	WheelB.ControlFeedbackSign := 1.0;
	WheelB.CarouselSign := -1.0;
	WheelB.StandardSign := 1.0;
	WheelB.DriveWheel := FALSE;
	WheelB.InnerFlag := TRUE;
	WheelB.WheelDirection := -1.0;
	WheelB.IndependentWheels := TRUE;

	WheelC.ControlFeedbackSign := 1.0;
	WheelC.CarouselSign := 1.0;
	WheelC.StandardSign := -1.0;
	WheelC.DriveWheel := TRUE;
	WheelC.InnerFlag := TRUE;
	WheelC.WheelDirection := -1.0;
	WheelC.IndependentWheels := TRUE;

	WheelD.ControlFeedbackSign := 1.0;
	WheelD.CarouselSign := -1.0;
	WheelD.StandardSign := -1.0;
	WheelD.DriveWheel := TRUE;
	WheelD.InnerFlag := FALSE;
	WheelD.WheelDirection := 1.0;
	WheelD.IndependentWheels := TRUE;
{END_IF}

lFunctionalMode := cFunctionalModeAny;

lMode REF= lSteerMode4WS;

lTargetAngleUpdateTimer.Period := cTargetAngleUpdatePeriod;
lTargetAngleUpdateTimer.Enable := TRUE;
lTargetAngleUpdateTimer.initialize();

                
END_METHOD

METHOD operator
                  requestSteerMode(gSystemPrimary.UInterface.SteerModeRequest);

lInput.InputAsPercentage := gSystemPrimary.UInterface.Steer;
lInput.operator();

SUPER^.operator();

lZeroTargetAngleSwitch.Value := gSystemPrimary.UInterface.ZeroSteerTargetAngle;
lZeroTargetAngleSwitch.operator();

IF (lEnableRelativeSteering) THEN
	lRegisterActive := TRUE;

	IF ((lZeroTargetAngleSwitch.Value) AND (lEnableZeroTargetAngleSwitch)) THEN
		zeroTargetAngle();
	END_IF

	lTargetAngleShift := lInput.Value;
ELSE
	lRegisterActive := TRUE;
	
	IF (lZeroTargetAngleSwitch.Value) THEN
		gSystemPrimary.Active.registerActive();
	END_IF
	
	IF (gSystemPrimary.Active.Allow) THEN
		lRequestedAbsoluteTargetAngle := lInput.Value;
		
		IF (lRequestedAbsoluteTargetAngle>=Mode.SteerAngleMaximum) THEN
			lRequestedAbsoluteTargetAngle := Mode.SteerAngleMaximum;
		END_IF
		IF (lRequestedAbsoluteTargetAngle<=Mode.SteerAngleMinimum) THEN
			lRequestedAbsoluteTargetAngle := Mode.SteerAngleMinimum;
		END_IF
	
		lTargetAngleShift := (lRequestedAbsoluteTargetAngle - lTargetAngle.Value) * cSteerAbsoluteShiftFactor;
	ELSE
		lTargetAngleShift := 0.0;	
	END_IF
	
	IF (lTargetAngleShift<-1.0) THEN
		lTargetAngleShift := -1.0;
	END_IF
	IF (lTargetAngleShift>1.0) THEN
		lTargetAngleShift := 1.0;
	END_IF
END_IF

updateTargetAngle();
checkWheelStates();

lWheelA.operator();
lWheelB.operator();
lWheelC.operator();
lWheelD.operator();

IF (lStalledSubSystems) THEN
	IF (NOT(lStalledSubSystemsPrevious)) THEN
		lStallClearPreCondition := NOT(InputPresentAny);
		lStallClearPreConditionCleared := FALSE;
	END_IF
	
	lStalled := TRUE;
END_IF

IF (lStalled) THEN
	lStallClearPreConditionCleared := (((InputPresentAny) AND (lStallClearPreCondition)) OR
		((NOT(InputPresentAny)) AND (NOT(lStallClearPreCondition))));
		
	lStalled := (NOT((gSystemPrimary.Travel.InputPresentAny) OR
		((InputPresentAny) AND
		(lStallClearPreConditionCleared))));
END_IF

IF (NOT(lStalled)) THEN
	WheelA.Throttle.clearStalled();
	WheelB.Throttle.clearStalled();
	WheelC.Throttle.clearStalled();
	WheelD.Throttle.clearStalled();
END_IF

                
END_METHOD

METHOD requestSteerMode : t_steer_mode_diagnostic
  VAR_INPUT
    requestedSteerMode : t_steer_mode;
  END_VAR
  VAR
    angle : REAL;
  END_VAR
                  IF (requestedSteerMode=cSteerModeNone) THEN
	RETURN;
END_IF

lSteerModeDiagnostic := cSteerModeDiagnosticOK;

IF (Mode.matches(requestedSteerMode)) THEN
	// essentially re-initializes to this steering mode
	angle := Mode.getInitialTargetAngle(lTargetAngle.Value,requestedSteerMode);
	IF (lTargetAngle.Value<>angle) THEN
		lTargetAngle.Value := angle;
		
		lWheelA.ModeChange := TRUE;
		lWheelB.ModeChange := TRUE;
		lWheelC.ModeChange := TRUE;
		lWheelD.ModeChange := TRUE;
		
		IF (lEnableSequentialModeChange) THEN
			lWheelA.ModeChangeDisableControl := FALSE;
			lWheelB.ModeChangeDisableControl := TRUE;
			lWheelC.ModeChangeDisableControl := TRUE;
			lWheelD.ModeChangeDisableControl := TRUE;
		END_IF
	END_IF
	
	requestSteerMode := lSteerModeDiagnostic;
	RETURN;
END_IF

IF (NOT(checkModeEnabled(requestedSteerMode))) THEN
	lSteerModeDiagnostic := cSteerModeDiagnosticNotEnabled;
	//gMessageManager.register(lCode:=cMCAdviseSteerModeIllegalRequest);

	requestSteerMode := lSteerModeDiagnostic;
	RETURN;
END_IF
	
IF ((lEnableOperatingModeLockOnSteerModeChange) AND
	(gSystemPrimary.OperatingMode.lock(cOperatingModeLockPeriod)<>cOperatingModeLocked)) THEN
	lSteerModeDiagnostic := cSteerModeDiagnosticUnableToLockDrive;
	//gMessageManager.register(lCode:=cMCAdviseSteerModeUnableToLockDrive);
	
	requestSteerMode := lSteerModeDiagnostic;
	RETURN;
END_IF

lMode.leave();
lMode REF= getMode(requestedSteerMode);
lSteerModeDiagnostic := cSteerModeDiagnosticChanging;

lTargetAngle.Value := Mode.getInitialTargetAngle(0.0,requestedSteerMode);

lWheelA.ModeChange := TRUE;
lWheelB.ModeChange := TRUE;
lWheelC.ModeChange := TRUE;
lWheelD.ModeChange := TRUE;

IF (lEnableSequentialModeChange) THEN // foobar apollo issue remaining - not all wheels are moving at the same time during mode changes, but could be spurious due to stalling
	lWheelA.ModeChangeDisableControl := FALSE;
	lWheelB.ModeChangeDisableControl := TRUE;
	lWheelC.ModeChangeDisableControl := TRUE;
	lWheelD.ModeChangeDisableControl := TRUE;
END_IF

// checkWheelStates();

                
END_METHOD

METHOD setCarouselAngle
                  lCarouselAngle := ATAN(lSteerWheelBase/lSteerWheelTrack);

                
END_METHOD

METHOD toggleSteerMode
                  CASE lMode.Mode OF
	cSteerModeNone:
		requestSteerMode(cSteerMode4WS);
	cSteerMode4WS:
		requestSteerMode(cSteerModeLateral);
	cSteerModeLateral:
		requestSteerMode(cSteerModeCarousel);
	cSteerModeCarousel:
		requestSteerMode(cSteerMode4WS);
END_CASE

                
END_METHOD

METHOD updateTargetAngle
                  IF (lEnableUpdateTimer) THEN
	lTargetAngleUpdateTimer.operator();
	IF (NOT(lTargetAngleUpdateTimer.lExpired)) THEN
		RETURN;
	END_IF
	lTargetAngleUpdateTimer.reset();
END_IF

IF (lTargetAngleShift=0.0) THEN
	IF (lEnableDerivedTargetAngleIncrement) THEN
		lTargetAngleIncrementDerivedPost := lTargetAngleIncrementDerived;
		
		IF (((lTargetAngleIncrementDerived>0) AND
			(ABS(lCurrentPositiveDelta)>cSteerAngleMaxDerivedUpdateDelta)) OR
			((lTargetAngleIncrementDerived<0) AND
			(ABS(lCurrentNegativeDelta)>cSteerAngleMaxDerivedUpdateDelta))) THEN
			lTargetAngleIncrementDerivedPost := 0.0;
		END_IF
			
		lTargetAngle.Value := lTargetAngle.Value + lTargetAngleIncrementDerivedPost;

		//lTargetAngleIncrementDerived := 0.0;
	END_IF
ELSE
	lTargetAngleIncrement := 0;

	IF (lTargetAngleShift>0) THEN
		IF (ABS(lCurrentPositiveDelta)<cSteerAngleMaxUpdateDelta) THEN
			lTargetAngleIncrement := lTargetAngleShift*cSteerAngleThrottleIncrement + cSteerAngleDeltaGain*lCurrentNegativeDelta;
			lTargetAngleIncrement := MAX(0,lTargetAngleIncrement);
		ELSIF (gSystemPrimary.Travel.Stationary) THEN
			lTargetAngleIncrement := lStationaryTargetAngleIncrement;
		END_IF
	END_IF

	IF (lTargetAngleShift<0) THEN
		IF (ABS(lCurrentNegativeDelta)<cSteerAngleMaxUpdateDelta) THEN
			lTargetAngleIncrement := lTargetAngleShift*cSteerAngleThrottleIncrement + cSteerAngleDeltaGain*lCurrentPositiveDelta;
			lTargetAngleIncrement := MIN(0,lTargetAngleIncrement);
		ELSIF (gSystemPrimary.Travel.Stationary) THEN
			lTargetAngleIncrement := 0.0 - lStationaryTargetAngleIncrement;
		END_IF
	END_IF

	lTargetAngle.Value := lTargetAngle.Value + lTargetAngleIncrement;
END_IF

lEnableDerivedTargetAngleIncrement := FALSE;
lTargetAngleIncrementDerived := 0.0;

lTargetAngle.operator();

IF (lTargetAngle.Value>=Mode.SteerAngleMaximum) THEN
	lTargetAngle.Value := Mode.SteerAngleMaximum;
END_IF
IF (lTargetAngle.Value<=Mode.SteerAngleMinimum) THEN
	lTargetAngle.Value := Mode.SteerAngleMinimum;
END_IF

// foobar, gradually change speed with steering angle, especially in lateral mode

                
END_METHOD

METHOD zeroTargetAngle
                  gSystemPrimary.ProgrammedMovementControl.request(cProgMovCode_Steer_0);

// lTargetAngle.Value := 0;
lInputPresentAuxilliaryRequest := TRUE;
                
END_METHOD

PROPERTY CarouselAngle : REAL
GET
                    CarouselAngle := lCarouselAngle;
                  
END_GET
END_PROPERTY

(* {attribute 'monitoring' := 'call'} *)
PROPERTY CurrentAbsDelta : REAL
GET
                    CurrentAbsDelta := lCurrentAbsDelta;
                  
END_GET
END_PROPERTY

PROPERTY CurrentMode : t_steer_mode
GET
                    CurrentMode := lMode.Mode;


                  
END_GET
SET
                    requestSteerMode(CurrentMode);
                  
END_SET
END_PROPERTY

(* {attribute 'monitoring' := 'call'} *)
PROPERTY CurrentNegativeDelta : REAL
GET
                    CurrentNegativeDelta := lCurrentNegativeDelta;
                  
END_GET
END_PROPERTY

(* {attribute 'monitoring' := 'call'} *)
PROPERTY CurrentPositiveDelta : REAL
GET
                    CurrentPositiveDelta := lCurrentPositiveDelta;
                  
END_GET
END_PROPERTY

PROPERTY EnableDerivedTargetAngleIncrement : BOOL
GET
                    EnableDerivedTargetAngleIncrement := lEnableDerivedTargetAngleIncrement;
                  
END_GET
SET
                    lEnableDerivedTargetAngleIncrement := EnableDerivedTargetAngleIncrement;
                  
END_SET
END_PROPERTY

PROPERTY Mode : REFERENCE TO SteerMode
GET
                    Mode REF= lMode;

                  
END_GET
END_PROPERTY

PROPERTY ModeChange : BOOL
GET
                    ModeChange := lModeChange;
                  
END_GET
END_PROPERTY

(* {attribute 'monitoring' := 'call'} *)
PROPERTY OK : BOOL
GET
                    OK := ((lAdjustState>=cAdjustStateGood) OR
	(lAdjustState<=cAdjustStateAdjusting));
                  
END_GET
END_PROPERTY

PROPERTY Ready : BOOL
GET
                    Ready := lMode.ready(State);

                  
END_GET
END_PROPERTY

PROPERTY StallClearPreCondition : BOOL
GET
                    StallClearPreCondition := lStallClearPreCondition;

                  
END_GET
END_PROPERTY

PROPERTY StallClearPreConditionCleared : BOOL
GET
                    StallClearPreConditionCleared := lStallClearPreConditionCleared;

                  
END_GET
END_PROPERTY

PROPERTY Stalled : BOOL
GET
                    Stalled := lStalled;

                  
END_GET
END_PROPERTY

PROPERTY StalledSubSystems : BOOL
GET
                    StalledSubSystems := lStalledSubSystems;

                  
END_GET
END_PROPERTY

(* {attribute 'monitoring' := 'call'} *)
PROPERTY State : t_adjust_state
GET
                    State := lAdjustState;
                  
END_GET
END_PROPERTY

PROPERTY Stationary : BOOL
GET
                    Stationary := lStationary;

                  
END_GET
END_PROPERTY

PROPERTY SteerAngleMaximum : REAL
GET
                    SteerAngleMaximum := Mode.SteerAngleMaximum;
                  
END_GET
END_PROPERTY

PROPERTY SteerAngleMinimum : REAL
GET
                    SteerAngleMinimum := Mode.SteerAngleMinimum;
                  
END_GET
END_PROPERTY

PROPERTY SteerAnglePhysicalMaximum : REAL
GET
                    SteerAnglePhysicalMaximum := cSteerAnglePhysicalMaximum;
                  
END_GET
END_PROPERTY

PROPERTY SteerAnglePhysicalMinimum : REAL
GET
                    SteerAnglePhysicalMinimum := cSteerAnglePhysicalMinimum;
                  
END_GET
END_PROPERTY

PROPERTY SteerMode4WS : REFERENCE TO SteerMode4WS
GET
                    SteerMode4WS ref= lSteerMode4WS;
                  
END_GET
END_PROPERTY

PROPERTY SteerModeCarousel : REFERENCE TO SteerModeCarousel
GET
                    SteerModeCarousel ref= lSteerModeCarousel;
                  
END_GET
END_PROPERTY

(* {attribute 'monitoring' := 'call'} *)
PROPERTY SteerModeDiagnostic : t_steer_mode_diagnostic
GET
                    SteerModeDiagnostic := lSteerModeDiagnostic;
                  
END_GET
END_PROPERTY

PROPERTY SteerModeLateral : REFERENCE TO SteerModeLateral
GET
                    SteerModeLateral ref= lSteerModeLateral;
                  
END_GET
END_PROPERTY

PROPERTY SteerModeReconfigure : REFERENCE TO SteerModeReconfigure
GET
                    SteerModeReconfigure ref= lSteerModeReconfigure;
                  
END_GET
END_PROPERTY

PROPERTY SteerWheelBase : REAL
GET
                    SteerWheelBase := lSteerWheelBase;
                  
END_GET
SET
                    lSteerWheelBase := SteerWheelBase;
setCarouselAngle();

                  
END_SET
END_PROPERTY

PROPERTY SteerWheelTrack : REAL
GET
                    SteerWheelTrack := lSteerWheelTrack;
                  
END_GET
SET
                    lSteerWheelTrack := SteerWheelTrack;
setCarouselAngle();

                  
END_SET
END_PROPERTY

(* {attribute 'monitoring' := 'call'} *)
PROPERTY TargetAngle : REAL
GET
                    TargetAngle := lTargetAngle.Value;
                  
END_GET
END_PROPERTY

PROPERTY TargetAngleIncrement : REAL
GET
                    TargetAngleIncrement := lTargetAngleIncrement;
                  
END_GET
END_PROPERTY

PROPERTY TargetAngleIncrementDerived : REAL
GET
                    TargetAngleIncrementDerived := lTargetAngleIncrementDerived;
                  
END_GET
SET
                    lTargetAngleIncrementDerived := TargetAngleIncrementDerived;
                  
END_SET
END_PROPERTY

PROPERTY TargetAngleIncrementDerivedPost : REAL
GET
                    TargetAngleIncrementDerivedPost := lTargetAngleIncrementDerivedPost;
                  
END_GET
END_PROPERTY

PROPERTY TargetAngleObject : REFERENCE TO ValueObjectReal
GET
                    TargetAngleObject REF= lTargetAngle;

                  
END_GET
END_PROPERTY

PROPERTY TriggerZeroTargetAngle : BOOL
SET
                    IF (TriggerZeroTargetAngle) THEN
	zeroTargetAngle();
END_IF
                  
END_SET
END_PROPERTY

PROPERTY WheelA : REFERENCE TO SlewMovement
GET
                    WheelA REF= lWheelA;

                  
END_GET
END_PROPERTY

PROPERTY WheelB : REFERENCE TO SlewMovement
GET
                    WheelB REF= lWheelB;

                  
END_GET
END_PROPERTY

PROPERTY WheelC : REFERENCE TO SlewMovement
GET
                    WheelC REF= lWheelC;

                  
END_GET
END_PROPERTY

PROPERTY WheelD : REFERENCE TO SlewMovement
GET
                    WheelD REF= lWheelD;

                  
END_GET
END_PROPERTY
END_FUNCTION_BLOCK

FUNCTION_BLOCK SteerMovementElectric EXTENDS SteerMovement
  VAR
    _ThrottleA : ThrottleMotorWithFeedback;
    _ThrottleB : ThrottleMotorWithFeedback;
    _ThrottleC : ThrottleMotorWithFeedback;
    _ThrottleD : ThrottleMotorWithFeedback;
  END_VAR

            ;
          

METHOD initialize
                  lSteerWheelTrack := gSystemPrimary.LocalMachinePrimary.WheelTrack; //foobar move to calibrate()?
lSteerWheelBase := gSystemPrimary.LocalMachinePrimary.WheelBase;

_ThrottleA.Name := 'ThrottleA';
_ThrottleA.SubSystem := cSubsystemSteerA;
_ThrottleA.ControllerMotor REF= gSystemPrimary.CANOpenMasterDrivePrimary.SteerA;
_ThrottleA.PositionObject REF= gSystemPrimary.CANOpenMasterDrivePrimary.SteerAngleA.AngleObject;
_ThrottleA.VelocityObject REF= gSystemPrimary.CANOpenMasterDrivePrimary.SteerAngleB.AngularVelocityObject;
WheelA.initializeSlew(_ThrottleA,gSystemPrimary.CANOpenMasterDrivePrimary.SteerAngleA,THIS^,gSystemPrimary.Travel);
registerNonOperational(ADR(_ThrottleA));

_ThrottleB.Name := 'ThrottleB';
_ThrottleB.SubSystem := cSubsystemSteerB;
_ThrottleB.ControllerMotor REF= gSystemPrimary.CANOpenMasterDrivePrimary.SteerB;
_ThrottleB.PositionObject REF= gSystemPrimary.CANOpenMasterDrivePrimary.SteerAngleB.AngleObject;
_ThrottleB.VelocityObject REF= gSystemPrimary.CANOpenMasterDrivePrimary.SteerAngleB.AngularVelocityObject;
WheelB.initializeSlew(_ThrottleB,gSystemPrimary.CANOpenMasterDrivePrimary.SteerAngleB,THIS^,gSystemPrimary.Travel);
registerNonOperational(ADR(_ThrottleB));

_ThrottleC.Name := 'ThrottleC';
_ThrottleC.SubSystem := cSubsystemSteerC;
_ThrottleC.ControllerMotor REF= gSystemPrimary.CANOpenMasterDrivePrimary.SteerC;
_ThrottleC.PositionObject REF= gSystemPrimary.CANOpenMasterDrivePrimary.SteerAngleC.AngleObject;
_ThrottleC.VelocityObject REF= gSystemPrimary.CANOpenMasterDrivePrimary.SteerAngleC.AngularVelocityObject;
WheelC.initializeSlew(_ThrottleC,gSystemPrimary.CANOpenMasterDrivePrimary.SteerAngleC,THIS^,gSystemPrimary.Travel);
registerNonOperational(ADR(_ThrottleC));

_ThrottleD.Name := 'ThrottleD';
_ThrottleD.SubSystem := cSubsystemSteerD;
_ThrottleD.ControllerMotor REF= gSystemPrimary.CANOpenMasterDrivePrimary.SteerD;
_ThrottleD.PositionObject REF= gSystemPrimary.CANOpenMasterDrivePrimary.SteerAngleD.AngleObject;
_ThrottleD.VelocityObject REF= gSystemPrimary.CANOpenMasterDrivePrimary.SteerAngleD.AngularVelocityObject;
WheelD.initializeSlew(_ThrottleD,gSystemPrimary.CANOpenMasterDrivePrimary.SteerAngleD,THIS^,gSystemPrimary.Travel);
registerNonOperational(ADR(_ThrottleD));

SUPER^.initialize();

lRegisterUMFSPrimary := TRUE;
lRegisterUMFSAuxilliary := TRUE;
lRegisterUMFSSecondary := TRUE;

lRegisterActive := TRUE;
lRegisterOperatingMode := TRUE;
	
lEnabled := TRUE;
lEnableOperatingModeSlow := FALSE;
lEnableOnlyOnActiveAllow := FALSE;
lEnableUMFSCheck := TRUE;
                
END_METHOD

PROPERTY DerivedThrottleA : REFERENCE TO ThrottleMotor
GET
                    DerivedThrottleA ref= _ThrottleA;
                  
END_GET
END_PROPERTY

PROPERTY DerivedThrottleB : REFERENCE TO ThrottleMotor
GET
                    DerivedThrottleB ref= _ThrottleB;
                  
END_GET
END_PROPERTY

PROPERTY DerivedThrottleC : REFERENCE TO ThrottleMotor
GET
                    DerivedThrottleC ref= _ThrottleC;
                  
END_GET
END_PROPERTY

PROPERTY DerivedThrottleD : REFERENCE TO ThrottleMotor
GET
                    DerivedThrottleD ref= _ThrottleD;
                  
END_GET
END_PROPERTY

PROPERTY TypeToken : t_medium_string
GET
                    TypeToken := 'mSteerElec';
                  
END_GET
END_PROPERTY
END_FUNCTION_BLOCK

FUNCTION_BLOCK Throttle EXTENDS OperationalParticleSet
  VAR
    lThrottle : REFERENCE TO ValueObjectPercentage;
    lValue : t_percentage;
    lSign : t_percentage := 1.0;
    lCurrentVelocity : REAL;
    lStationary : BOOL;
    lStalled : BOOL;
  END_VAR

            ;
          

METHOD clearStalled
                  lStalled := false;
                
END_METHOD

METHOD initialize
                  IF (NOT(__ISVALIDREF(lThrottle))) THEN
	gCodeErrorHandler(pMessage:=CONCAT('null reference in ',lIdentity));
END_IF

SUPER^.initialize();

lCurrentVelocity := 0.0;
lStationary := FALSE;
lStalled := FALSE;

                
END_METHOD

METHOD operator
                  lThrottle.Value := lValue * lSign;

SUPER^.operator();

                
END_METHOD

PROPERTY CurrentDirection : t_direction
GET
                    IF (CurrentVelocity=0) THEN
	CurrentDirection := cDirectionStationary;
ELSIF (CurrentVelocity>0.0) THEN
	CurrentDirection := cDirectionForward;
ELSE
	CurrentDirection := cDirectionReverse;
END_IF
                  
END_GET
END_PROPERTY

PROPERTY CurrentVelocity : REAL
GET
                    CurrentVelocity := lCurrentVelocity;
                  
END_GET
END_PROPERTY

PROPERTY Sign : t_percentage
GET
                    Sign := lSign;
                  
END_GET
SET
                    lSign := Sign;
                  
END_SET
END_PROPERTY

PROPERTY Stalled : BOOL
GET
                    Stalled := lStalled;

                  
END_GET
END_PROPERTY

PROPERTY Stationary : BOOL
GET
                    Stationary := lStationary;

                  
END_GET
END_PROPERTY

PROPERTY Throttle : REFERENCE TO ValueObjectPercentage
GET
                    Throttle ref= lThrottle;
                  
END_GET
SET
                    lThrottle REF= Throttle;

                  
END_SET
END_PROPERTY

PROPERTY TypeToken : t_medium_string
GET
                    TypeToken := 'Throttle';
                  
END_GET
END_PROPERTY

(* {attribute 'monitoring' := 'call'} *)
PROPERTY Value : t_percentage
GET
                    Value := lValue;
                  
END_GET
SET
                    lValue := Value;
                  
END_SET
END_PROPERTY
END_FUNCTION_BLOCK

FUNCTION_BLOCK ThrottleDerived EXTENDS Throttle
  VAR
    lMovement : REFERENCE TO Movement;
    _Throttle : ValueObjectPercentage;
  END_VAR

            ;
          

METHOD initialize
                  lThrottle REF= _Throttle;
_Throttle.initializeValueObjectOp(OpSelf,'Value','Throttle value','',cValueStyleConfigurable);

IF (NOT(__ISVALIDREF(lMovement))) THEN
	gCodeErrorHandler(pMessage:=CONCAT('null reference in ',lIdentity));
END_IF

SUPER^.initialize();


                
END_METHOD

METHOD operator
                  SUPER^.operator();

lMovement.InputSecondaryValue := lThrottle.Value;

                
END_METHOD

PROPERTY Movement : REFERENCE TO Movement
GET
                    Movement ref= lMovement;
                  
END_GET
SET
                    lMovement ref= Movement;
                  
END_SET
END_PROPERTY

PROPERTY TypeToken : t_medium_string
GET
                    TypeToken := 'ThrottleDeriv';
                  
END_GET
END_PROPERTY
END_FUNCTION_BLOCK

FUNCTION_BLOCK ThrottleMotor EXTENDS Throttle
  VAR
    lControllerMotor : REFERENCE TO ControllerMotor;
    _Throttle : ValueObjectPercentage;
  END_VAR

            ;
          

METHOD initialize
                  lThrottle REF= _Throttle;
_Throttle.initializeValueObjectOp(OpSelf,'Value','Throttle value','',cValueStyleConfigurable);

IF (NOT(__ISVALIDREF(lControllerMotor))) THEN
	gCodeErrorHandler(pMessage:=CONCAT('null reference in ',lIdentity));
END_IF

SUPER^.initialize();

                
END_METHOD

METHOD operator
                  SUPER^.operator();

lControllerMotor.RequestedThrottle := lThrottle.Value;

lCurrentVelocity := lControllerMotor.Velocity;
lStationary := lControllerMotor.Stationary;
lStalled := lControllerMotor.Stalled;

                
END_METHOD

PROPERTY ControllerMotor : REFERENCE TO ControllerMotor
GET
                    ControllerMotor REF= lControllerMotor;

                  
END_GET
SET
                    lControllerMotor ref= ControllerMotor;
                  
END_SET
END_PROPERTY

PROPERTY CurrentVelocity : REAL
GET
                    CurrentVelocity := lCurrentVelocity;
                  
END_GET
END_PROPERTY

PROPERTY TypeToken : t_medium_string
GET
                    TypeToken := 'ThrottleMotor';
                  
END_GET
END_PROPERTY
END_FUNCTION_BLOCK

FUNCTION_BLOCK ThrottleMotorWithFeedback EXTENDS ThrottleMotor
  VAR
    lPosition : REFERENCE TO ValueObjectReal;
    lVelocity : REFERENCE TO ValueObjectReal;
  END_VAR

            ;
          

METHOD operator
                  SUPER^.operator();

lCurrentVelocity := lVelocity.Value;
lStationary := ((lVelocity.Value=0) AND (lThrottle.Value=0));
lStalled := false;
                
END_METHOD

METHOD initialize
                  IF ((NOT(__ISVALIDREF(lPosition))) OR
	(NOT(__ISVALIDREF(lVelocity)))) THEN
	gCodeErrorHandler(pMessage:=CONCAT('null reference in ',lIdentity));
END_IF

SUPER^.initialize();

                
END_METHOD

PROPERTY PositionObject : REFERENCE TO ValueObjectReal
GET
                    PositionObject ref= lPosition;
                  
END_GET
SET
                    lPosition ref= PositionObject;
                  
END_SET
END_PROPERTY

PROPERTY TypeToken : t_medium_string
GET
                    TypeToken := 'ThrottleMotFdb';
                  
END_GET
END_PROPERTY

PROPERTY VelocityObject : REFERENCE TO ValueObjectReal
GET
                    VelocityObject ref= lVelocity;
                  
END_GET
SET
                    lVelocity ref= VelocityObject;
                  
END_SET
END_PROPERTY
END_FUNCTION_BLOCK

FUNCTION_BLOCK ThrottleVirtual EXTENDS Throttle
  VAR
    _Throttle : ValueObjectPercentage;
  END_VAR

            ;
          

METHOD initialize
                  lThrottle REF= _Throttle;
_Throttle.initializeValueObjectOp(OpSelf,'Value','Throttle value','',cValueStyleConfigurable);

SUPER^.initialize();


                
END_METHOD

PROPERTY TypeToken : t_medium_string
GET
                    TypeToken := 'ThrottleVirtual';
                  
END_GET
END_PROPERTY
END_FUNCTION_BLOCK

FUNCTION_BLOCK Alarm EXTENDS OutputSystemState
  VAR CONSTANT
    cSecondaryRequiredAvailability : t_percentage := 0.1;
  END_VAR
  VAR
    lAlarmSecondaryPowerFail : ReportableAlarmEscalating;
    lEnableAlarmInReverseOnly : BOOL := FALSE;
  END_VAR

            ;
          

METHOD initialize
                  Name := 'Alarm';

lAlarmSecondaryPowerFail.initializeState(NopSelf,'',cACSecondaryPowerFail);
lAlarmSecondaryPowerFail.Life := 10;
lAlarmSecondaryPowerFail.InitialSeverity := cSeverityNone;
lAlarmSecondaryPowerFail.SeverityWarningTimeout := T#1S;
lAlarmSecondaryPowerFail.SeverityErrorTimeout := T#2S;
lAlarmSecondaryPowerFail.SeverityCriticalTimeout := T#5S;

lOutputSystemState := cSystemStateOperational;

SUPER^.initialize();
SubSystem := cSubsystemPowerpack;

                
END_METHOD

METHOD operator
                  IF (lEnableAlarmInReverseOnly) THEN
	lOutput.Value := (gSystemPrimary.Travel.Throttle.Value < 0);
ELSE
	lOutput.Value := gSystemPrimary.OperatingMode.Moving;
END_IF

IF ((lOutput.Value) AND
	(gSystemPrimary.lSecondaryPowerSupply.Availability<cSecondaryRequiredAvailability)) THEN	
	lAlarmSecondaryPowerFail.trigger(FALSE);
	
	lOutput.Value := FALSE;
END_IF

SUPER^.operator();


                
END_METHOD
END_FUNCTION_BLOCK

FUNCTION_BLOCK Beacons EXTENDS OutputSystemState
  VAR CONSTANT
    cSecondaryRequiredAvailability : t_percentage := 0.1;
  END_VAR
  VAR
    lAlarmSecondaryPowerFail : ReportableAlarmEscalating;
  END_VAR

            ;
          

METHOD initialize
                  Name := 'Beacons';

lAlarmSecondaryPowerFail.initializeState(NopSelf,'',cACBeaconsSecondaryPowerFail);
lAlarmSecondaryPowerFail.Life := 10;
lAlarmSecondaryPowerFail.InitialSeverity := cSeverityNone;
lAlarmSecondaryPowerFail.SeverityWarningTimeout := T#1S;
lAlarmSecondaryPowerFail.SeverityErrorTimeout := T#2S;
lAlarmSecondaryPowerFail.SeverityCriticalTimeout := T#5S;

SUPER^.initialize();
SubSystem := cSubsystemBeacons;

lOutputSystemState := cSystemStateOperational;
                
END_METHOD

METHOD operator
                  lOutput.Value := (gSystemPrimary.SystemState.State=cSystemStateOperational);

IF ((lOutput.Value) AND
	(gSystemPrimary.lSecondaryPowerSupply.Availability<cSecondaryRequiredAvailability)) THEN	
	lAlarmSecondaryPowerFail.trigger(FALSE);
	
	lOutput.Value := FALSE;
END_IF

SUPER^.operator();



                
END_METHOD
END_FUNCTION_BLOCK

FUNCTION_BLOCK CabinSecondaryPower EXTENDS OutputSystemStateAuto

            ;
          

METHOD initialize
                  Name := 'CabinSecPwr';

SUPER^.initialize();
SubSystem := cSubsystemPowerpack;

lOutputSystemState := cSystemStatePreparing;

                
END_METHOD
END_FUNCTION_BLOCK

FUNCTION_BLOCK EstopLoad EXTENDS OutputSystemStateAuto

            ;
          

METHOD initialize
                  Name := 'EstopLoad';

SUPER^.initialize();
SubSystem := cSubsystemUInterface;

lOutputSystemState := cSystemStatePoweringUp;

                
END_METHOD
END_FUNCTION_BLOCK

FUNCTION_BLOCK Horn EXTENDS OutputSystemState

            ;
          

METHOD initialize
                  Name := 'Horn';

SUPER^.initialize();
SubSystem := cSubsystemPowerpack;

lOutputSystemState := cSystemStatePreOperational;
                
END_METHOD

METHOD operator
                  lOutput.Value := gSystemPrimary.UInterface.Horn;

SUPER^.operator();

                
END_METHOD
END_FUNCTION_BLOCK

FUNCTION_BLOCK Lights EXTENDS OutputSystemState

            ;
          

METHOD initialize
                  Name := 'Lights';

SUPER^.initialize();
SubSystem := cSubsystemLights;

lOutputSystemState := cSystemStateCharging;
                
END_METHOD

METHOD initializeLights
                  
                
END_METHOD
END_FUNCTION_BLOCK

FUNCTION_BLOCK PumpCooling EXTENDS OutputSystemState

            ;
          

METHOD initialize
                  Name := 'PumpCooling';

SUPER^.initialize();
SubSystem := cSubsystemBattery;

lOutputSystemState := cSystemStateOperational;
                
END_METHOD

METHOD operator
                  lOutput.Value := (gSystemPrimary.SystemState.State=cSystemStateOperational);

SUPER^.operator();

                
END_METHOD

METHOD initializePumpCooling
                  
                
END_METHOD
END_FUNCTION_BLOCK

FUNCTION_BLOCK SensorSupply EXTENDS OutputSystemStateAuto

            ;
          

METHOD initialize
                  Name := 'SensorSupply';

SUPER^.initialize();
SubSystem := cSubsystemPowerpack;

lOutputSystemState := cSystemStatePreparing;

lOutput.Scaling := 12000;
                
END_METHOD

METHOD initializeSensorSupply
                  
                
END_METHOD
END_FUNCTION_BLOCK

FUNCTION_BLOCK SecondaryPowerSupplyPrimary EXTENDS SecondaryPowerSupply

            ;
          

METHOD initialize
                  lControllerSecondaryPowerSupplyA REF= gSystemPrimary.CANOpenMasterSystemPrimary.SecondaryPowerSupplyA;
lControllerSecondaryPowerSupplyB REF= gSystemPrimary.CANOpenMasterSystemPrimary.SecondaryPowerSupplyB;

SUPER^.initialize();



                
END_METHOD

PROPERTY BMSConnected : BOOL
GET
                    BMSConnected := (gSystemPrimary.BMS.CurrentState>=cBMSStateConnected);
                  
END_GET
END_PROPERTY
END_FUNCTION_BLOCK

FUNCTION_BLOCK ActiveSystem EXTENDS Active
  VAR CONSTANT
    cActiveExitOperationalTimeout : t_time := TIME#10m0s0ms;
  END_VAR
  VAR
    lVREnableExitOperational : ValueReferenceBool;
    lEnableExitOperational : BOOL := TRUE;
    lCausalStopOnTimeout : ReportableSystemControl;
    lExitOperationalTimer : t_timer;
    lRegisterUI : BOOL := FALSE;
    lValueUI : BOOL := FALSE;
  END_VAR

            ;
          

METHOD initialize
                  Name := 'Active';

lVREnableExitOperational.initializeValueReference(lEnableExitOperational,NopSelf,'EnblExitOp','Automatically exit operational upon timeout','',cValueStyleParameter);

lCausalStopOnTimeout.initializeState(NopSelf,'',cCCStopOnTimeout);
lCausalStopOnTimeout.Control := cSystemControlStop;
lCausalStopOnTimeout.AllowableSystemState := cSystemStatePreOperational;

SUPER^.initialize();

lExitOperationalTimer.lEnable := TRUE;
lExitOperationalTimer.lPeriod := cActiveExitOperationalTimeout;
lExitOperationalTimer.initialize();

{IF defined(target_d19)}
lPreTimer.lPeriod := T#750MS;
lPostTimer.lPeriod := T#5S;
{END_IF}
                
END_METHOD

METHOD operator
                  lValueUI := lRegisterUI;
lRegisterUI := FALSE;

IF (gSystemPrimary.UInterface.UMFS) THEN
	registerActive();
END_IF

SUPER^.operator();

IF (gSystemPrimary.SystemState.State<>cSystemStateOperational) THEN
	lState := t_active_state.cActiveStateNone;
	lExitOperationalTimer.reset();
END_IF

IF (IsActive) THEN
	lExitOperationalTimer.reset();
END_IF
lExitOperationalTimer.operator();

IF ((gSystemPrimary.SystemState.State=cSystemStateOperational) AND
	((lExitOperationalTimer.lExpired) AND (lEnableExitOperational))) THEN
	lCausalStopOnTimeout.trigger(FALSE);
END_IF

                
END_METHOD

METHOD registerUI
                  lRegisterUI := TRUE;
                
END_METHOD

PROPERTY ExitOperationalPeriod : t_time
GET
                    ExitOperationalPeriod := lExitOperationalTimer.Period;
                  
END_GET
SET
                    lExitOperationalTimer.Period := ExitOperationalPeriod;
                  
END_SET
END_PROPERTY

PROPERTY IsActive : BOOL
GET
                    IsActive := ((lState<>t_active_state.cActiveStateNone) OR (lValueUI));

                  
END_GET
END_PROPERTY

PROPERTY PumpRunning : BOOL
GET
                    PumpRunning := lAllowPreCondition;

                  
END_GET
SET
                    lAllowPreCondition := PumpRunning;
                  
END_SET
END_PROPERTY

PROPERTY TypeToken : t_medium_string
GET
                    TypeToken := 'ActiveSystem';
                  
END_GET
END_PROPERTY
END_FUNCTION_BLOCK

FUNCTION_BLOCK OperatingMode EXTENDS NonOperationalParticleSet
  VAR
    lCausalWaitingForParked : ReportableCausal;
    lVRForceSlow : ValueReferenceBool;
    lForceSlow : BOOL := FALSE;
    lMode : t_operating_mode := cOperatingModeInoperable;
    lEnableAutoUnpark : BOOL := TRUE;
    lSlow : BOOL := FALSE;
    lAllStopped : BOOL := TRUE;
    lAllParked : BOOL := TRUE;
    lAnyStalled : BOOL := FALSE;
    lSlowFactor : REAL := 1.0;
    lLockTimer : t_timer;
    lEnableLockTimer : BOOL := FALSE;
  END_VAR

            ;
          

METHOD initialize
                  Name := 'OperatingMode';

lCausalWaitingForParked.initializeState(NopSelf,'',cCCWaitingForParked);

lVRForceSlow.initializeValueReference(lForceSlow,NopSelf,'ForceSlow','Force slow mode','',cValueStyleParameter);

SUPER^.initialize();

lSlow := FALSE;

lAllParked := TRUE;
lAllStopped := TRUE;
lAnyStalled := FALSE;

lMode := cOperatingModeParked;

lLockTimer.Enable := TRUE;
lLockTimer.Period := T#1S;
lLockTimer.initialize();

                
END_METHOD

METHOD inoperable : t_operating_mode
                  lMode := cOperatingModeInoperable;

inoperable := lMode;

                
END_METHOD

METHOD lock : t_operating_mode
  VAR_INPUT
    period : t_time;
  END_VAR
                  IF (lMode=cOperatingModeStopped) THEN
	lMode := cOperatingModeLocked;
	IF (period>T#0S) THEN
		lLockTimer.Period := period;
		lLockTimer.reset();
		lEnableLockTimer := TRUE;
	ELSE
		lEnableLockTimer := FALSE;		
	END_IF
END_IF

lock := lMode;

                
END_METHOD

METHOD normal
                  lSlow := FALSE;
                
END_METHOD

METHOD operator
  VAR
    lOverrideValue : INT;
  END_VAR
                  request(gSystemPrimary.UInterface.OperatingMethodRequest);

IF (gSystemPrimary.SystemState.State<cSystemStateOperational) THEN
	park();
END_IF

IF (gSystemPrimary.SystemState.State<=cSystemStatePreOperational) THEN
	reset();
END_IF

IF ((lEnableAutoUnpark) AND
	(gSystemPrimary.SystemState.State=cSystemStateOperational) AND
	(lMode<=cOperatingModeParking)) THEN
	unpark();
END_IF

(* wait until movement has stopped *)
IF (gSystemPrimary.SystemState.State=cSystemStateExitOperational) THEN
	IF (lMode>cOperatingModeParked) THEN
		gSystemPrimary.SystemState.transitionAllowDown(cSystemStateExitOperational,ADR(lCausalWaitingForParked),lCausalWaitingForParked.Override);
	END_IF
END_IF

IF ((lMode=cOperatingModeParking) AND (lAllParked)) THEN
	lMode := cOperatingModeParked;
END_IF

IF ((lMode=cOperatingModeUnparking) AND (lAllStopped)) THEN
	lMode := cOperatingModeStopped;
END_IF

IF ((lEnableLockTimer) AND (lMode=cOperatingModeLocked)) THEN
	lLockTimer.operator();
	IF (lLockTimer.Expired) THEN
		unlock();
	END_IF
END_IF

IF (lMode>cOperatingModeLocked) THEN
	IF (lAllStopped) THEN
		lMode := cOperatingModeStopped;
	ELSIF (lAnyStalled) THEN
		lMode := cOperatingModeStalled;
	ELSIF ((lSlow) OR
		(lForceSlow)) THEN
		lMode := cOperatingModeSlow;
	ELSE
		lMode := cOperatingModeNormal;
	END_IF
END_IF

lAllParked := TRUE;
lAllStopped := TRUE;
lAnyStalled := FALSE;

                
END_METHOD

METHOD park : t_operating_mode
                  (* allows recovery from inoperable and locked *)

IF (lMode=cOperatingModeParked) THEN
	RETURN;
END_IF

lMode := cOperatingModeParking;

park := lMode;

                
END_METHOD

METHOD registerReady
                  ;
(*lAllParked := ((lAllParked) AND (TRUE));
lAllStopped := ((lAllStopped) AND (TRUE));*)
                
END_METHOD

METHOD registerRunning
                  lAllStopped := FALSE;
lAllParked := FALSE;
                
END_METHOD

METHOD registerStalled
                  lAnyStalled := TRUE;
lAllStopped := FALSE;
lAllParked := FALSE;
                
END_METHOD

METHOD registerStopped
                  lAllStopped := ((lAllStopped) AND (TRUE));
                
END_METHOD

METHOD registerUnParked
                  lAllParked := FALSE;

                
END_METHOD

METHOD request
  VAR_INPUT
    requestedOperatingMethod : t_operating_method;
  END_VAR
                  
                
END_METHOD

METHOD reset
                  lSlow := FALSE;
lMode := cOperatingModeParked;
                
END_METHOD

METHOD slow
                  lSlow := TRUE;
                
END_METHOD

METHOD togglePark : t_operating_mode
                  IF ((lMode=cOperatingModeParked) OR
	(lMode=cOperatingModeParking)) THEN
	lMode := cOperatingModeUnparking;
	togglePark := lMode;
	RETURN;
END_IF

lMode := cOperatingModeParking;

togglePark := lMode;

                
END_METHOD

METHOD toggleSpeed : t_operating_mode
                  lSlow := NOT(lSlow);

                
END_METHOD

METHOD unlock : t_operating_mode
                  lMode := cOperatingModeStopped;

unLock := lMode;

                
END_METHOD

METHOD unpark : t_operating_mode
                  IF ((lMode=cOperatingModeParked) OR
	(lMode=cOperatingModeParking)) THEN
	lMode := cOperatingModeUnparking;
END_IF

unpark := lMode;

                
END_METHOD

PROPERTY IsSlow : BOOL
GET
                    IsSlow := (lMode=cOperatingModeSlow);

                  
END_GET
END_PROPERTY

PROPERTY LockedOrParked : BOOL
GET
                    LockedOrParked := (lMode<=cOperatingModeLocked);
                  
END_GET
END_PROPERTY

PROPERTY Mode : t_operating_mode
GET
                    Mode := lMode;
                  
END_GET
END_PROPERTY

PROPERTY Moving : BOOL
GET
                    Moving := (lMode>cOperatingModeStopped);
                  
END_GET
END_PROPERTY

PROPERTY Ready : BOOL
GET
                    Ready := (lMode>=cOperatingModeStopped);
                  
END_GET
END_PROPERTY

PROPERTY SlowFactor : REAL
GET
                    SlowFactor := lSlowFactor;

                  
END_GET
END_PROPERTY

PROPERTY Stopped : BOOL
GET
                    Stopped := (lMode<=cOperatingModeStopped);
                  
END_GET
END_PROPERTY

PROPERTY TypeToken : t_medium_string
GET
                    TypeToken := 'OperatingMode';
                  
END_GET
END_PROPERTY
END_FUNCTION_BLOCK

FUNCTION_BLOCK PeripheralPrimary EXTENDS Peripheral
  VAR
    lAlarmSoftware : ReportableAlarm;
    lAlarmConfiguration : ReportableAlarm;
    lAlarmVBBS : ReportableAlarm;
    lAlarmVBB1 : ReportableAlarm;
    lAlarmVBB2 : ReportableAlarm;
    lAlarmPLCTemp : ReportableAlarm;
  END_VAR

            ;
          

METHOD initialize
                  lAlarmSoftware.initializeState(NopSelf,'',cACSoftware);
lAlarmConfiguration.initializeState(NopSelf,'',cACConfiguration);

lAlarmVBBS.initializeState(NopSelf,'VBBS',cACVoltage);
lAlarmVBB1.initializeState(NopSelf,'VBB1',cACVoltage);
lAlarmVBB2.initializeState(NopSelf,'VBB2',cACVoltage);
lAlarmPLCTemp.initializeState(NopSelf,'',cACTemperature);

SUPER^.initialize();

registerReportable(ADR(lAlarmSoftware),cRCSoftware);
registerReportable(ADR(lAlarmConfiguration),cRCConfiguration);

registerReportable(ADR(lAlarmVBBS),cRCVBBS);
registerReportable(ADR(lAlarmVBB1),cRCVBB1);
registerReportable(ADR(lAlarmVBB2),cRCVBB2);
registerReportable(ADR(lAlarmPLCTemp),cRCPLCTemp);
                
END_METHOD

METHOD operator
                  SUPER^.operator();

(* traffic FROM master PLC *)

lExternalState := fMergeBitsIntoWord(pWord:=lExternalState,pData:=gSystemPrimary.SystemState.State,pStart:=0);
lExternalState := fMergeBitsIntoWord(pWord:=lExternalState,pData:=gSystemPrimary.OperatingMode.Mode,pStart:=4);
lExternalState := fMergeBoolIntoWord(pWord:=lExternalState,pData:=gSystemPrimary.lUMFS.Allow,pStart:=8);

(* traffic to master PLC *)

IF (lOperatingModeLockRequest.Value) THEN
	gSystemPrimary.OperatingMode.lock(T#2S);
END_IF

IF (lOperatingModeRunningRegister.Value) THEN
	gSystemPrimary.OperatingMode.registerRunning();
ELSE
	gSystemPrimary.OperatingMode.registerStopped();
END_IF

IF (lUMFSRegister.Value) THEN
	gSystemPrimary.lUMFS.registerSlave();
END_IF

                
END_METHOD
END_FUNCTION_BLOCK

FUNCTION_BLOCK UIEvent EXTENDS NonOperationalParticleSet
  VAR
    lCausalCommandStart : ReportableCausal;
    lCausalCommandStop : ReportableCausal;
    lUIEventCode : t_ui_event_code := cUIEventCodeNone;
    lUIEventCodePrevious : t_ui_event_code := cUIEventCodeNone;
  END_VAR

            ;
          

METHOD _operator
                  CASE lUIEventCode OF
	cUIEventCodeToggleLights:
		gSystemPrimary.Lights.toggleOutput();
		
	cUIEventCodeStart:
		IF (gSystemPrimary.SystemState.State=cSystemStatePreOperational) THEN
			lCausalCommandStart.trigger(FALSE);
			gSystemPrimary.SystemState.transitionStart(cSystemStateOperational,ADR(lCausalCommandStart),lCausalCommandStart.Override);
		END_IF
		
	cUIEventCodeStop:
		IF (gSystemPrimary.SystemState.State>cSystemStatePreOperational) THEN
			lCausalCommandStop.trigger(FALSE);
			gSystemPrimary.SystemState.transitionStop(cSystemStatePreOperational,ADR(lCausalCommandStop),lCausalCommandStop.Override);
		END_IF
END_CASE

                
END_METHOD

METHOD initialize
                  Name := 'UIEvent';

lCausalCommandStart.initializeState(NopSelf,'',cCCCommandStart);
lCausalCommandStop.initializeState(NopSelf,'',cCCCommandStop);

SUPER^.initialize();

                
END_METHOD

METHOD operator
                  lUIEventCode := gSystemPrimary.UInterface.UIEventCodeRequest;

IF (lUIEventCode=lUIEventCodePrevious) THEN
	RETURN;
END_IF
lUIEventCodePrevious := lUIEventCode;

IF (lUIEventCode=cUIEventCodeNone) THEN
	RETURN;
END_IF

_operator();

                
END_METHOD

PROPERTY TypeToken : t_medium_string
GET
                    TypeToken := 'UIEvent';
                  
END_GET
END_PROPERTY
END_FUNCTION_BLOCK

FUNCTION_BLOCK UMFS EXTENDS OperationalParticleSet
  VAR_INPUT
    lEnableSwitch : BOOL := TRUE;  (* UInterface *)
    lEnableSeat : BOOL := FALSE;  (* deprecated *)
    lEnableSignal : BOOL := TRUE;  (* not used *)
    lEnablePrimary : BOOL := FALSE;  (* primary movement - should be false *)
    lEnableSecondary : BOOL := TRUE;  (* automation - prog mov *)
    lEnableAuxilliary : BOOL := TRUE;  (* automation - zero target angle *)
    lEnableSlave : BOOL := FALSE;  (* slave - via UInterface *)
  END_VAR
  VAR CONSTANT
    cSmoothingPeriod : t_time := TIME#2s0ms;  (* foobar *)
  END_VAR
  VAR
    lAllow : ValueObjectBool;
    lSmoothingTimer : t_timer;
    lSeatSwitch : BOOL;
    lUISwitch : BOOL;
    lUISignal : BOOL;
    lUIPrimary : BOOL;
    lUISecondary : BOOL;
    lUIAuxilliary : BOOL;
    lUISlave : BOOL;
  END_VAR

            ;
          

METHOD initialize
                  Name := 'UMFS';

lAllow.initializeValueObjectOp(OpSelf,'Allow','UMFS allows related movements','',cValueStyleConfigurable);

SUPER^.initialize();
SubSystem := cSubsystemUInterface;

lSeatSwitch := FALSE;
lUISwitch := FALSE;
lUISignal := FALSE;
lUIPrimary := FALSE;
lUIAuxilliary := FALSE;
lUISlave := FALSE;

lSmoothingTimer.Enable := TRUE;
lSmoothingTimer.Period := cSmoothingPeriod;
lSmoothingTimer.initialize();

                
END_METHOD

METHOD operator
                  IF (gSystemPrimary.UInterface.UMFS) THEN
	registerUISwitch();
END_IF

lAllow.Value := (((lSeatSwitch) AND (lUISignal) AND (lEnableSeat)) OR
	((lUISwitch) AND (lEnableSwitch)) OR
	((lUISignal) AND (lEnableSignal)) OR
	((lUIPrimary) AND (lEnablePrimary)) OR
	((lUISecondary) AND (lEnableSecondary)) OR
	((lUIAuxilliary) AND (lEnableAuxilliary)) OR
	((lUISlave) AND (lEnableSlave)));

lSmoothingTimer.operator();
IF (lAllow.Value) THEN
	lSmoothingTimer.reset();
END_IF
lAllow.Value := ((lAllow.Value) OR (NOT(lSmoothingTimer.Expired)));

SUPER^.operator();

lSeatSwitch := FALSE;
lUISwitch := FALSE;
lUISignal := FALSE;
lUIPrimary := FALSE;
lUISecondary := FALSE;
lUIAuxilliary := FALSE;
lUISlave := FALSE;
                
END_METHOD

METHOD registerSeat
                  lSeatSwitch := TRUE;

                
END_METHOD

METHOD registerSlave
                  lUISlave := true;
                
END_METHOD

METHOD registerUIAuxilliary
                  lUIAuxilliary := TRUE;
                
END_METHOD

METHOD registerUIPrimary
                  lUIPrimary := TRUE;
                
END_METHOD

METHOD registerUISecondary
                  lUISecondary := TRUE;
                
END_METHOD

METHOD registerUISignal
                  lUISignal := TRUE;

                
END_METHOD

METHOD registerUISwitch
                  lUISwitch := TRUE;

                
END_METHOD

PROPERTY Allow : BOOL
GET
                    Allow := lAllow.Value;

                  
END_GET
END_PROPERTY

PROPERTY TypeToken : t_medium_string
GET
                    TypeToken := 'UMFS';
                  
END_GET
END_PROPERTY
END_FUNCTION_BLOCK

FUNCTION_BLOCK UInterfaceCabin EXTENDS UInterfacePLC
  VAR CONSTANT
    cTelescopingDeadband : t_percentage := 0.1;
  END_VAR
  VAR
    lControllerUInterfaceCabin : REFERENCE TO ControllerUInterfaceCabin;
  END_VAR

            ;
          

METHOD initialize
                  Name := 'Cabin';

IF (NOT(__ISVALIDREF(lControllerUInterfaceCabin))) THEN
	gCodeErrorHandler(pMessage:=CONCAT('null reference in ',lIdentity));
END_IF

SUPER^.initialize();

lUInterfaceId := t_ui_id.cUIIdA;



                
END_METHOD

METHOD initializeUInterfaceCabin
  VAR_INPUT
    controllerUInterfaceCabin : REFERENCE TO ControllerUInterfaceCabin;
  END_VAR
                  lControllerUInterfaceCabin REF= controllerUInterfaceCabin;

                
END_METHOD

PROPERTY AutomationStart : BOOL
GET
                    AutomationStart := FALSE;

IF ((Active) AND
	(gSystemPrimary.ProgrammedMovementControl.Enabled)) THEN
	AutomationStart := lControllerUInterfaceCabin.AutomationStart;
END_IF

                  
END_GET
END_PROPERTY

PROPERTY Horn : BOOL
GET
                    Horn := lControllerUInterfaceCabin.Horn; 
                  
END_GET
END_PROPERTY

PROPERTY TwistlockLock : BOOL
GET
                    TwistlockLock := FALSE;

IF (Active) THEN
	TwistlockLock := lControllerUInterfaceCabin.TwistlockLock;
END_IF
                  
END_GET
END_PROPERTY

PROPERTY TwistlockUnlock : BOOL
GET
                    TwistlockUnlock := FALSE;

IF (Active) THEN
	TwistlockUnlock := lControllerUInterfaceCabin.TwistlockUnlock;
END_IF

                  
END_GET
END_PROPERTY

PROPERTY ZeroSteerTargetAngle : BOOL
GET
                    ZeroSteerTargetAngle := FALSE;

IF (Active) THEN
	ZeroSteerTargetAngle := lControllerUInterfaceCabin.ZeroSteerTargetAngle;
END_IF

                  
END_GET
END_PROPERTY

PROPERTY Estop : BOOL
GET
                    Estop := lControllerUInterfaceCabin.Estop;
                  
END_GET
END_PROPERTY

PROPERTY IsSlow : BOOL
GET
                    IsSlow := FALSE;

                  
END_GET
END_PROPERTY

(* {attribute 'monitoring' := 'call'} *)
PROPERTY JoystickInputPresent : BOOL
GET
                    JoystickInputPresent := lControllerUInterfaceCabin.JoystickInputPresent;

                  
END_GET
END_PROPERTY

PROPERTY Lift : t_percentage
GET
                    Lift := 0;

IF (Active) THEN
	Lift := lControllerUInterfaceCabin.Lift;
END_IF

                  
END_GET
END_PROPERTY

PROPERTY LiftBalanceAB : t_percentage
GET
                    LiftBalanceAB := 0;

IF (Active) THEN
	LiftBalanceAB := lControllerUInterfaceCabin.LiftBalanceAB;
END_IF


                  
END_GET
END_PROPERTY

PROPERTY LiftBalanceAD : t_percentage
GET
                    LiftBalanceAD := 0;

IF (Active) THEN
	LiftBalanceAD := lControllerUInterfaceCabin.LiftBalanceAD;
END_IF


                  
END_GET
END_PROPERTY

(* {attribute 'monitoring' := 'call'} *)
PROPERTY LiftJoystickInputPresent : BOOL
GET
                    LiftJoystickInputPresent := lControllerUInterfaceCabin.LiftJoystickInputPresent;

                  
END_GET
END_PROPERTY

PROPERTY SideshiftAB : t_percentage
GET
                    SideshiftAB := 0;

IF (Active) THEN
	SideshiftAB := lControllerUInterfaceCabin.SideshiftAB;
END_IF

                  
END_GET
END_PROPERTY

PROPERTY SideshiftCD : t_percentage
GET
                    SideshiftCD := 0;

IF (Active) THEN
	SideshiftCD := lControllerUInterfaceCabin.SideshiftCD;
END_IF

                  
END_GET
END_PROPERTY

PROPERTY SpreaderTelescopingExtend : BOOL
GET
                    SpreaderTelescopingExtend := FALSE;

IF ((Active) AND
	(gSystemPrimary.FunctionalModeControl.CurrentMode=cFunctionalModeSpreaderConfiguration)) THEN
	SpreaderTelescopingExtend := lControllerUInterfaceCabin.SpreaderTelescopingExtend;
END_IF


                  
END_GET
END_PROPERTY

PROPERTY SpreaderTelescopingRetract : BOOL
GET
                    SpreaderTelescopingRetract := FALSE;

IF ((Active) AND
	(gSystemPrimary.FunctionalModeControl.CurrentMode=cFunctionalModeSpreaderConfiguration)) THEN
	SpreaderTelescopingRetract := lControllerUInterfaceCabin.SpreaderTelescopingRetract;
END_IF
                  
END_GET
END_PROPERTY

PROPERTY Steer : t_percentage
GET
                    Steer := 0;

IF (Active) THEN
	Steer := lControllerUInterfaceCabin.Steer;
END_IF
                  
END_GET
END_PROPERTY

PROPERTY Stop : BOOL
GET
                    Stop := lControllerUInterfaceCabin.Stop;

                  
END_GET
END_PROPERTY

PROPERTY Topbeam : t_percentage
GET
                    Topbeam := 0;

IF ((Active) AND
	(gSystemPrimary.FunctionalModeControl.CurrentMode=cFunctionalModeTopbeamConfiguration) AND
	(gSystemPrimary.FunctionalModeControl.Active)) THEN
	Topbeam := lControllerUInterfaceCabin.Topbeam;
END_IF

                  
END_GET
END_PROPERTY

(* {attribute 'monitoring' := 'call'} *)
PROPERTY Travel : t_percentage
GET
                    Travel := 0;

IF (Active) THEN
	Travel := lControllerUInterfaceCabin.Travel;
END_IF



                  
END_GET
END_PROPERTY

(* {attribute 'monitoring' := 'call'} *)
PROPERTY TravelJoystickInputPresent : BOOL
GET
                    TravelJoystickInputPresent := FALSE;

IF (Active) THEN
	TravelJoystickInputPresent := lControllerUInterfaceCabin.TravelJoystickInputPresent;
END_IF

                  
END_GET
END_PROPERTY

PROPERTY TypeToken : t_medium_string
GET
                    TypeToken := 'UICabin';
                  
END_GET
END_PROPERTY

PROPERTY UMFS : BOOL
GET
                    UMFS := FALSE;

IF (Active) THEN
	UMFS := lControllerUInterfaceCabin.UMFS;
END_IF

                  
END_GET
END_PROPERTY

PROPERTY Emgy : BOOL
GET
                    Emgy := lControllerUInterfaceCabin.Emgy;

                  
END_GET
END_PROPERTY

PROPERTY EnableBatteryPack : BOOL
GET
                    EnableBatteryPack := lControllerUInterfaceCabin.EnableBatteryPack;

                  
END_GET
END_PROPERTY
END_FUNCTION_BLOCK

FUNCTION_BLOCK PackMovementPLC EXTENDS PackMovement

            
          

METHOD read
                  lSteerStateA := gSystemPrimary.Steering.WheelA.State;
lSteerStateB := gSystemPrimary.Steering.WheelB.State;
lSteerStateC := gSystemPrimary.Steering.WheelC.State;
lSteerStateD := gSystemPrimary.Steering.WheelD.State;

lSteerTargetAngle := gSystemPrimary.Steering.TargetAngle;
lSteerCurrentMode := gSystemPrimary.Steering.CurrentMode;
	
lTravelActive := gSystemPrimary.Travel.Active;
lTravelVelocity := gSystemPrimary.Travel.ThrottleValue;

lLiftActive := gSystemPrimary.Lift.Active;
lLiftABPosition := 0.0;
lLiftCDPosition := 0.0;

lProgrammedMovementCurrent := gSystemPrimary.ProgrammedMovementControl.CurrentMovement;
lProgrammedMovementState := gSystemPrimary.ProgrammedMovementControl.CurrentState;

                
END_METHOD
END_FUNCTION_BLOCK

FUNCTION_BLOCK PackReportablePLC EXTENDS PackReportable
  VAR
    lReportableChannelUIR : REFERENCE TO ReportableChannelUIR;
    lReportedCount : UINT := 0;
    a : USINT := 0;
    b : USINT := 0;
    c : USINT := 0;
    d : USINT := 0;
    e : USINT := 0;
  END_VAR

            
          

METHOD read
  VAR
    reportable : POINTER TO t_ui_reportable;
  END_VAR
                  lReportableA.valid := FALSE;
lReportableB.valid := FALSE;
lReportableC.valid := FALSE;
lReportableD.valid := FALSE;

a := a+ 1;

reportable := lReportableChannelUIR.popOrCycle();
IF (reportable=0) THEN
b := b+ 1;
	RETURN;
END_IF
lReportableA := reportable^;
lReportedCount := lReportedCount + 1;

reportable := lReportableChannelUIR.popOrCycle();
IF (reportable=0) THEN
c := c+ 1;
	RETURN;
END_IF
lReportableB := reportable^;
lReportedCount := lReportedCount + 1;

reportable := lReportableChannelUIR.popOrCycle();
IF (reportable=0) THEN
d := d+ 1;
	RETURN;
END_IF
lReportableC := reportable^;
lReportedCount := lReportedCount + 1;

reportable := lReportableChannelUIR.popOrCycle();
IF (reportable=0) THEN
e := e+ 1;
	RETURN;
END_IF
lReportableD := reportable^;
lReportedCount := lReportedCount + 1;

                
END_METHOD

METHOD initialize
                  IF (NOT(__ISVALIDREF(lReportableChannelUIR))) THEN
	gCodeErrorHandler(pMessage:='null reference in PackReportablePLC');
END_IF

SUPER^.initialize();

                
END_METHOD

METHOD initializePackReportablePLC
  VAR_INPUT
    reportableChannelUIR : REFERENCE TO ReportableChannelUIR;
  END_VAR
                  lReportableChannelUIR ref= reportableChannelUIR;
                
END_METHOD
END_FUNCTION_BLOCK

FUNCTION_BLOCK PackSystemPLC EXTENDS PackSystem
  VAR
    lUInterface : REFERENCE TO UInterface;
  END_VAR

            
          

METHOD read
                  lFunctionalMode := gSystemPrimary.FunctionalModeControl.CurrentMode;
lToggle := gSystemPrimary.Cycle.Toggle;
lSystemState := gSystemPrimary.SystemState.State;
lOperatingMode := gSystemPrimary.OperatingMode.Mode;
lSpeedModeSlow := FALSE;
lLightStatus := gSystemPrimary.Lights.OutputObject.Value;

lUIReady := lUInterface.Ready;
lUIModeRequest := lUInterface.UIModeRequest;
lUIMode := lUInterface.UIMode;

lHours := REAL_TO_UINT(gSystemPrimary.Cycle.OperationalHours);
lSOC := gSystemPrimary.BMS.SOC;
lCurrent := gSystemPrimary.BMS.Current;

lInputMode := lUInterface.InputMode;
lUIOrientation := lUInterface.UIOrientation;

lAvailability := gSystemPrimary.BMS.Availability;

                
END_METHOD

METHOD initializePackSystemPLC
  VAR_INPUT
    uInterface : REFERENCE TO UInterface;
  END_VAR
                  lUInterface ref= uInterface;
                
END_METHOD

METHOD initialize
                  IF (NOT(__ISVALIDREF(lUInterface))) THEN
	gCodeErrorHandler(pMessage:='null reference in PackSystemPLC');
END_IF

SUPER^.initialize();

                
END_METHOD
END_FUNCTION_BLOCK

FUNCTION_BLOCK PackUICommandPLC EXTENDS PackUICommand
  VAR
    lUInterface : REFERENCE TO UInterfacePLC;
  END_VAR

            
          

METHOD initializePackUICommandPLC
  VAR_INPUT
    uInterface : REFERENCE TO UInterfacePLC;
  END_VAR
                  lUInterface ref= uInterface;
                
END_METHOD

METHOD initialize
                  IF (NOT(__ISVALIDREF(lUInterface))) THEN
	gCodeErrorHandler(pMessage:='null reference in PackUICommandPLC');
END_IF

SUPER^.initialize();

                
END_METHOD

METHOD write
  VAR
    reportable : POINTER TO t_ui_reportable;
  END_VAR
                  lUInterface.UIEventCodeRequest := lUIEventCodeRequest;
lUInterface.SteerModeRequest := lSteerModeRequest;
lUInterface.OperatingMethodRequest := lOperatingMethodRequest;
lUInterface.FunctionalModeRequest := lFunctionalModeRequest;
lUInterface.AutomationRequest := lAutomationRequest;

lUInterface.UIModeResponse := lUIModeResponse;
lUInterface.InputMode := lInputModeRequest;
lUInterface.UIOrientation := lUIOrientationRequest;
lUInterface.IsBeginner := lIsBeginner;

IF (fCheckUIRValidity(lReportableA)) THEN
	lUInterface.UIRRouter.reportUIR(lReportableA);
END_IF

IF (fCheckUIRValidity(lReportableB)) THEN
	lUInterface.UIRRouter.reportUIR(lReportableB);
END_IF

                
END_METHOD
END_FUNCTION_BLOCK

FUNCTION_BLOCK PackChannelUInterfacePLC EXTENDS PackChannelUInterface

            ;
          

METHOD pullPLCIncomingChannel : BOOL
                  pullPLCIncomingChannel := FALSE;

lPackProvider.pull();

IF (lPLCIncomingPacket.Byte1<>lPackProvider.PackIn1) THEN
	lPLCIncomingPacket.Byte1 := lPackProvider.PackIn1;
	lPLCIncomingPacket.Byte1 := lPLCIncomingPacket.Byte1 OR INT_TO_USINT(cPackCodeUICommand);
	gSystemPrimary.Active.registerUI();
	pullPLCIncomingChannel := TRUE;
END_IF

IF (lPLCIncomingPacket.Byte2<>lPackProvider.PackIn2) THEN
	lPLCIncomingPacket.Byte2 := lPackProvider.PackIn2;
	gSystemPrimary.Active.registerUI();
	pullPLCIncomingChannel := TRUE;
END_IF

IF (lPLCIncomingPacket.Byte3<>lPackProvider.PackIn3) THEN
	lPLCIncomingPacket.Byte3 := lPackProvider.PackIn3;
	gSystemPrimary.Active.registerUI();
	pullPLCIncomingChannel := TRUE;
END_IF

IF (lPLCIncomingPacket.Byte4<>lPackProvider.PackIn4) THEN
	lPLCIncomingPacket.Byte4 := lPackProvider.PackIn4;
	gSystemPrimary.Active.registerUI();
	pullPLCIncomingChannel := TRUE;
END_IF

IF (lPLCIncomingPacket.Byte5<>lPackProvider.PackIn5) THEN
	lPLCIncomingPacket.Byte5 := lPackProvider.PackIn5;
	gSystemPrimary.Active.registerUI();
	pullPLCIncomingChannel := TRUE;
END_IF

IF (lPLCIncomingPacket.Byte6<>lPackProvider.PackIn6) THEN
	lPLCIncomingPacket.Byte6 := lPackProvider.PackIn6;
	gSystemPrimary.Active.registerUI();
	pullPLCIncomingChannel := TRUE;
END_IF

IF (lPLCIncomingPacket.Byte7<>lPackProvider.PackIn7) THEN
	lPLCIncomingPacket.Byte7 := lPackProvider.PackIn7;
	gSystemPrimary.Active.registerUI();
	pullPLCIncomingChannel := TRUE;
END_IF

IF (lPLCIncomingPacket.Byte8<>lPackProvider.PackIn8) THEN
	lPLCIncomingPacket.Byte8 := lPackProvider.PackIn8;
	gSystemPrimary.Active.registerUI();
	pullPLCIncomingChannel := TRUE;
END_IF

                
END_METHOD

METHOD pushPLCOutgoingChannel
                  lPackProvider.PackOut1 := lPLCOutgoingPacket.Byte1;
lPackProvider.PackOut2 := lPLCOutgoingPacket.Byte2;
lPackProvider.PackOut3 := lPLCOutgoingPacket.Byte3;
lPackProvider.PackOut4 := lPLCOutgoingPacket.Byte4;
lPackProvider.PackOut5 := lPLCOutgoingPacket.Byte5;
lPackProvider.PackOut6 := lPLCOutgoingPacket.Byte6;
lPackProvider.PackOut7 := lPLCOutgoingPacket.Byte7;
lPackProvider.PackOut8 := lPLCOutgoingPacket.Byte8;

lPackProvider.push();

                
END_METHOD

METHOD operator
                  lPackTimer.operator();
IF ((NOT(lPackTimer.Enable)) OR (lPackTimer.Expired)) THEN
	lPackTimer.reset();

	lPLCOutgoingChannel.pack(lPLCOutgoingPacket);
	pushPLCOutgoingChannel();
			
	IF (lDebugPack) THEN
		lDebugPackPacket.copy(lPLCOutgoingPacket);
	END_IF
END_IF

IF (pullPLCIncomingChannel()) THEN
	IF (lDebugUnpack) THEN
		lDebugUnpackPacket.copy(lPLCIncomingPacket);
	END_IF

	lPLCIncomingChannel.unpack(lPLCIncomingPacket);
END_IF

                
END_METHOD
END_FUNCTION_BLOCK

FUNCTION_BLOCK PackChannelUInterfacePLCorig EXTENDS PackChannelUInterface
  VAR
    lControllerUInterface : REFERENCE TO ControllerUInterface;
  END_VAR

            ;
          

METHOD initialize
                  IF (NOT(__ISVALIDREF(lControllerUInterface))) THEN
	gCodeErrorHandler(pMessage:=CONCAT('null reference in ',lIdentity));
END_IF

SUPER^.initialize();


                
END_METHOD

METHOD pullPLCIncomingChannel : BOOL
                  pullPLCIncomingChannel := FALSE;

IF (lPLCIncomingPacket.Byte1<>lControllerUInterface.PackIn1) THEN
	lPLCIncomingPacket.Byte1 := lControllerUInterface.PackIn1;
	lPLCIncomingPacket.Byte1 := lPLCIncomingPacket.Byte1 OR INT_TO_USINT(cPackCodeUICommand);
	gSystemPrimary.Active.registerUI();
	pullPLCIncomingChannel := TRUE;
END_IF

IF (lPLCIncomingPacket.Byte2<>lControllerUInterface.PackIn2) THEN
	lPLCIncomingPacket.Byte2 := lControllerUInterface.PackIn2;
	gSystemPrimary.Active.registerUI();
	pullPLCIncomingChannel := TRUE;
END_IF

IF (lPLCIncomingPacket.Byte3<>lControllerUInterface.PackIn3) THEN
	lPLCIncomingPacket.Byte3 := lControllerUInterface.PackIn3;
	gSystemPrimary.Active.registerUI();
	pullPLCIncomingChannel := TRUE;
END_IF

IF (lPLCIncomingPacket.Byte4<>lControllerUInterface.PackIn4) THEN
	lPLCIncomingPacket.Byte4 := lControllerUInterface.PackIn4;
	gSystemPrimary.Active.registerUI();
	pullPLCIncomingChannel := TRUE;
END_IF

IF (lPLCIncomingPacket.Byte5<>lControllerUInterface.PackIn5) THEN
	lPLCIncomingPacket.Byte5 := lControllerUInterface.PackIn5;
	gSystemPrimary.Active.registerUI();
	pullPLCIncomingChannel := TRUE;
END_IF

IF (lPLCIncomingPacket.Byte6<>lControllerUInterface.PackIn6) THEN
	lPLCIncomingPacket.Byte6 := lControllerUInterface.PackIn6;
	gSystemPrimary.Active.registerUI();
	pullPLCIncomingChannel := TRUE;
END_IF

IF (lPLCIncomingPacket.Byte7<>lControllerUInterface.PackIn7) THEN
	lPLCIncomingPacket.Byte7 := lControllerUInterface.PackIn7;
	gSystemPrimary.Active.registerUI();
	pullPLCIncomingChannel := TRUE;
END_IF

IF (lPLCIncomingPacket.Byte8<>lControllerUInterface.PackIn8) THEN
	lPLCIncomingPacket.Byte8 := lControllerUInterface.PackIn8;
	gSystemPrimary.Active.registerUI();
	pullPLCIncomingChannel := TRUE;
END_IF

                
END_METHOD

METHOD pushPLCOutgoingChannel
                  lControllerUInterface.PackOut1 := lPLCOutgoingPacket.Byte1;
lControllerUInterface.PackOut2 := lPLCOutgoingPacket.Byte2;
lControllerUInterface.PackOut3 := lPLCOutgoingPacket.Byte3;
lControllerUInterface.PackOut4 := lPLCOutgoingPacket.Byte4;
lControllerUInterface.PackOut5 := lPLCOutgoingPacket.Byte5;
lControllerUInterface.PackOut6 := lPLCOutgoingPacket.Byte6;
lControllerUInterface.PackOut7 := lPLCOutgoingPacket.Byte7;
lControllerUInterface.PackOut8 := lPLCOutgoingPacket.Byte8;

                
END_METHOD

METHOD operator
                  lPackTimer.operator();
IF ((NOT(lPackTimer.Enable)) OR (lPackTimer.Expired)) THEN
	lPackTimer.reset();

	lPLCOutgoingChannel.pack(lPLCOutgoingPacket);
	pushPLCOutgoingChannel();
			
	IF (lDebugPack) THEN
		lDebugPackPacket.copy(lPLCOutgoingPacket);
	END_IF
END_IF

IF (pullPLCIncomingChannel()) THEN
	IF (lDebugUnpack) THEN
		lDebugUnpackPacket.copy(lPLCIncomingPacket);
	END_IF

	lPLCIncomingChannel.unpack(lPLCIncomingPacket);
END_IF

                
END_METHOD

METHOD initializePackChannelUInterfacePLC
  VAR_INPUT
    packSystem : REFERENCE TO PackSystemPLC;
    packMovement : REFERENCE TO PackMovementPLC;
    packReportable : REFERENCE TO PackReportablePLC;
    packSpreader : REFERENCE TO PackSpreader;
    packUICommand : REFERENCE TO PackUICommandPLC;
    controllerUInterface : REFERENCE TO ControllerUInterface;
    uInterface : REFERENCE TO UInterfacePLC;
  END_VAR
                  lControllerUInterface REF= controllerUInterface;

initializePackChannelUInterface(packSystem,
	packMovement,
	packReportable,
	packSpreader,
	packUICommand);

packSystem.initializePackSystemPLC(uInterface);
packUICommand.initializePackUICommandPLC(controllerUInterface,
	uInterface);

                
END_METHOD
END_FUNCTION_BLOCK

FUNCTION_BLOCK UInterfaceRadio EXTENDS UInterfacePLC
  VAR CONSTANT
    cTelescopingDeadband : t_percentage := 0.1;
  END_VAR
  VAR
    lVREnableUIOrientation : ValueReferenceBool;
    lEnableUIOrientation : BOOL := TRUE;
    lInputEstopStatus : ValueObjectBoolInputReferenceDINTFiltered;
    lInputSafetyHardwiredA : ValueObjectBoolInputReferenceDINTAsBool;
    lInputSafetyHardwiredB : ValueObjectBoolInputReferenceDINTAsBool;  (* foobar changes to wiring harness *)
    lPower : OutputSystemStateAuto;
    lControllerUInterfaceRadio : REFERENCE TO ControllerUInterfaceRadio;
    lInputMode : t_input_mode;
    lUIOrientation : t_ui_orientation := cUIOrientationForward;
    lSlowFactor : REAL := 1.0;
  END_VAR

            ;
          

METHOD initialize
                  Name := 'Radio';

IF (NOT(__ISVALIDREF(lControllerUInterfaceRadio))) THEN
	gCodeErrorHandler(pMessage:=CONCAT('null reference in ',lIdentity));
END_IF

lVREnableUIOrientation.initializeValueReference(lEnableUIOrientation,NopSelf,'EnblOrientation','Enable control of UI orientation','',cValueStyleParameter);

lInputEstopStatus.initializeValueObjectOp(OpSelf,'EstopStatus','Radio estop status','',cValueStyleConfigurable);
lInputSafetyHardwiredA.initializeValueObjectOp(OpSelf,'SafetyStatusA','Radio safety status A','',cValueStyleConfigurable);
lInputSafetyHardwiredB.initializeValueObjectOp(OpSelf,'SafetyStatusB','Radio safety status B','',cValueStyleConfigurable);

lPower.Name := 'Power';
registerOperational(ADR(lPower));

SUPER^.initialize();

lUInterfaceId := t_ui_id.cUIIdA;

lPower.OutputSystemState := cSystemStatePreparing;

lInputEstopStatus.FilterEnabled := TRUE; //foobar usually false for RadioB
lInputEstopStatus.Period := T#100MS;

                
END_METHOD

METHOD operator
                  IF (gSystemPrimary.SystemState.State<cSystemStateOperational) THEN
	lInputMode := cInputModeDefault;
END_IF

SUPER^.operator();

                
END_METHOD

METHOD initializeUInterfaceRadio
  VAR_INPUT
    controllerUInterfaceRadio : REFERENCE TO ControllerUInterfaceRadio;
  END_VAR
                  lControllerUInterfaceRadio REF= controllerUInterfaceRadio;

                
END_METHOD

METHOD initializeUInterfaceRadioIO
  VAR_INPUT
    outputRadio : REFERENCE TO DINT;
    inputEstopStatus : REFERENCE TO DINT;
    inputUMFSA : REFERENCE TO DINT;
    inputUMFSB : REFERENCE TO DINT;
  END_VAR
                  lPower.initializeOutput(outputRadio);
	
lInputEstopStatus.InputReference REF= inputEstopStatus;

lInputSafetyHardwiredA.InputReference REF= inputUMFSA;
lInputSafetyHardwiredB.InputReference REF= inputUMFSB;

                
END_METHOD

PROPERTY AutomationStart : BOOL
GET
                    AutomationStart := FALSE;

IF ((Active) AND
	(gSystemPrimary.ProgrammedMovementControl.Enabled)) THEN
	AutomationStart := lControllerUInterfaceRadio.AutomationStart;
END_IF

                  
END_GET
END_PROPERTY

PROPERTY Emgy : BOOL
GET
                    Emgy := lControllerUInterfaceRadio.Emgy;

                  
END_GET
END_PROPERTY

PROPERTY Horn : BOOL
GET
                    Horn := lControllerUInterfaceRadio.Horn; 
                  
END_GET
END_PROPERTY

PROPERTY TwistlockLock : BOOL
GET
                    TwistlockLock := FALSE;

IF (Active) THEN
	TwistlockLock := lControllerUInterfaceRadio.TwistlockLock;
END_IF
                  
END_GET
END_PROPERTY

PROPERTY Estop : BOOL
GET
                    Estop := lInputEstopStatus.Value;
                  
END_GET
END_PROPERTY

PROPERTY InputMode : t_input_mode
GET
                    InputMode := lInputMode;

                  
END_GET
SET
                    IF ((InputMode<>cInputModeNone) AND (gSystemPrimary.SystemState.State=cSystemStateOperational)) THEN
	lInputMode := InputMode;
END_IF

                  
END_SET
END_PROPERTY

PROPERTY InputSafetyHardwiredAObject : REFERENCE TO ValueObjectBool
GET
                    InputSafetyHardwiredAObject REF= lInputSafetyHardwiredA;

                  
END_GET
END_PROPERTY

PROPERTY InputSafetyHardwiredBObject : REFERENCE TO ValueObjectBool
GET
                    InputSafetyHardwiredBObject REF= lInputSafetyHardwiredB;

                  
END_GET
END_PROPERTY

PROPERTY IsSlow : BOOL
GET
                    IsSlow := TRUE;

                  
END_GET
END_PROPERTY

(* {attribute 'monitoring' := 'call'} *)
PROPERTY JoystickInputPresent : BOOL
GET
                    JoystickInputPresent := lControllerUInterfaceRadio.JoystickInputPresent;

                  
END_GET
END_PROPERTY

PROPERTY Lift : t_percentage
GET
                    Lift := 0;

IF ((Active) AND
	(gSystemPrimary.FunctionalModeControl.CurrentMode<>cFunctionalModeTopbeamConfiguration) AND
	(InputMode=cInputModeDefault)) THEN
	Lift := lControllerUInterfaceRadio.RightRotation;
END_IF

                  
END_GET
END_PROPERTY

PROPERTY LiftBalanceAB : t_percentage
GET
                    LiftBalanceAB := 0;

IF (Active) THEN
	CASE lUIOrientation OF
		cUIOrientationForward:
			LiftBalanceAB := lControllerUInterfaceRadio.RightXaxis;

		cUIOrientationSide:
			LiftBalanceAB := lControllerUInterfaceRadio.RightYaxis;

		cUIOrientationReverse:
			LiftBalanceAB := lControllerUInterfaceRadio.RightXaxis * -1.0;

		cUIOrientationOpposite:		
			LiftBalanceAB := lControllerUInterfaceRadio.RightYaxis * -1.0;
	END_CASE
END_IF

                  
END_GET
END_PROPERTY

PROPERTY LiftBalanceAD : t_percentage
GET
                    LiftBalanceAD := 0;

IF (Active) THEN
	CASE lUIOrientation OF
		cUIOrientationForward:
			LiftBalanceAD := lControllerUInterfaceRadio.RightYaxis;

		cUIOrientationSide:
			LiftBalanceAD := lControllerUInterfaceRadio.RightXaxis;

		cUIOrientationReverse:
			LiftBalanceAD := lControllerUInterfaceRadio.RightYaxis * -1.0;

		cUIOrientationOpposite:		
			LiftBalanceAD := lControllerUInterfaceRadio.RightXaxis * -1.0;
	END_CASE
END_IF


                  
END_GET
END_PROPERTY

(* {attribute 'monitoring' := 'call'} *)
PROPERTY LiftJoystickInputPresent : BOOL
GET
                    LiftJoystickInputPresent := lControllerUInterfaceRadio.RightJoystickInputPresent;

                  
END_GET
END_PROPERTY

PROPERTY SafetyCANOpen : BOOL
GET
                    SafetyCANOpen := lControllerUInterfaceRadio.SafetyCANOpen;

                  
END_GET
END_PROPERTY

PROPERTY Sideshift : t_percentage
GET
                    Sideshift := 0;

IF (Active) THEN
	CASE lUIOrientation OF
		cUIOrientationForward:
			Sideshift := lControllerUInterfaceRadio.RightXaxis;

		cUIOrientationSide:
			Sideshift := lControllerUInterfaceRadio.RightYaxis;

		cUIOrientationReverse:
			Sideshift := lControllerUInterfaceRadio.RightXaxis * -1.0;

		cUIOrientationOpposite:		
			Sideshift := lControllerUInterfaceRadio.RightYaxis * -1.0;
	END_CASE
END_IF
                  
END_GET
END_PROPERTY

PROPERTY SideshiftAB : t_percentage
GET
                    SideshiftAB := 0;

SideshiftAB := Sideshift;
IF (SideshiftBalanceAD<0.0) THEN
	SideshiftAB := Sideshift * ABS(1.0+SideshiftBalanceAD);
END_IF

                  
END_GET
END_PROPERTY

PROPERTY SideshiftBalanceAD : t_percentage
GET
                    SideshiftBalanceAD := 0;

IF (Active) THEN
	CASE lUIOrientation OF
		cUIOrientationForward:
			SideshiftBalanceAD := lControllerUInterfaceRadio.RightYaxis;

		cUIOrientationSide:
			SideshiftBalanceAD := lControllerUInterfaceRadio.RightXaxis;

		cUIOrientationReverse:
			SideshiftBalanceAD := lControllerUInterfaceRadio.RightYaxis * -1.0;

		cUIOrientationOpposite:		
			SideshiftBalanceAD := lControllerUInterfaceRadio.RightXaxis * -1.0;
	END_CASE
END_IF
                  
END_GET
END_PROPERTY

PROPERTY SideshiftCD : t_percentage
GET
                    SideshiftCD := 0;

SideshiftCD := Sideshift;
IF (SideshiftBalanceAD>0.0) THEN
	SideshiftCD := Sideshift * ABS(1.0-SideshiftBalanceAD);
END_IF

                  
END_GET
END_PROPERTY

PROPERTY SlowFactor : REAL
GET
                    SlowFactor := lSlowFactor;

                  
END_GET
SET
                    lSlowFactor := SlowFactor;
                  
END_SET
END_PROPERTY

PROPERTY SpreaderTelescopingExtend : BOOL
GET
                    SpreaderTelescopingExtend := FALSE;

IF ((Active) AND
	(gSystemPrimary.FunctionalModeControl.CurrentMode<>cFunctionalModeTopbeamConfiguration) AND
	(InputMode=cInputModeSpreaderConfiguration)) THEN
	SpreaderTelescopingExtend := (lControllerUInterfaceRadio.RightRotation>cTelescopingDeadband);
END_IF


                  
END_GET
END_PROPERTY

PROPERTY SpreaderTelescopingRetract : BOOL
GET
                    SpreaderTelescopingRetract := FALSE;

IF ((Active) AND
	(gSystemPrimary.FunctionalModeControl.CurrentMode<>cFunctionalModeTopbeamConfiguration) AND
	(InputMode=cInputModeSpreaderConfiguration)) THEN
	SpreaderTelescopingRetract := (lControllerUInterfaceRadio.RightRotation<(-cTelescopingDeadband));
END_IF
                  
END_GET
END_PROPERTY

PROPERTY Steer : t_percentage
GET
                    Steer := 0;

IF ((Active) AND
	(gSystemPrimary.FunctionalModeControl.CurrentMode<>cFunctionalModeTopbeamConfiguration) AND
	(InputMode=cInputModeDefault)) THEN
	
	CASE lUIOrientation OF
		cUIOrientationForward:
			Steer := lControllerUInterfaceRadio.LeftXaxis;

		cUIOrientationSide:
			Steer := lControllerUInterfaceRadio.LeftYaxis;

		cUIOrientationReverse:
			Steer := lControllerUInterfaceRadio.LeftXaxis * -1.0;

		cUIOrientationOpposite:		
			Steer := lControllerUInterfaceRadio.LeftYaxis * -1.0;
	END_CASE
END_IF
                  
END_GET
END_PROPERTY

PROPERTY Stop : BOOL
GET
                    Stop := ((lControllerUInterfaceRadio.Stop) AND
	(NOT(lControllerUInterfaceRadio.TimedStop)));

                  
END_GET
END_PROPERTY

PROPERTY Topbeam : t_percentage
GET
                    Topbeam := 0;

IF ((Active) AND
	(gSystemPrimary.FunctionalModeControl.CurrentMode=cFunctionalModeTopbeamConfiguration) AND
	(gSystemPrimary.FunctionalModeControl.Active) AND
	(InputMode=cInputModeTopbeamConfiguration)) THEN
	Topbeam := lControllerUInterfaceRadio.RightRotation;
END_IF
                  
END_GET
END_PROPERTY

(* {attribute 'monitoring' := 'call'} *)
PROPERTY Travel : t_percentage
GET
                    Travel := 0;

IF ((Active) AND
	(gSystemPrimary.FunctionalModeControl.CurrentMode<>cFunctionalModeTopbeamConfiguration) AND
	(InputMode=cInputModeDefault)) THEN
	
	CASE lUIOrientation OF
		cUIOrientationForward:
			Travel := lControllerUInterfaceRadio.LeftYaxis;

		cUIOrientationSide:
			Travel := lControllerUInterfaceRadio.LeftXaxis * -1.0;

		cUIOrientationReverse:
			Travel := lControllerUInterfaceRadio.LeftYaxis * -1.0;

		cUIOrientationOpposite:		
			Travel := lControllerUInterfaceRadio.LeftXaxis;
	END_CASE
END_IF



                  
END_GET
END_PROPERTY

(* {attribute 'monitoring' := 'call'} *)
PROPERTY TravelJoystickInputPresent : BOOL
GET
                    TravelJoystickInputPresent := lControllerUInterfaceRadio.LeftJoystickInputPresent;

                  
END_GET
END_PROPERTY

PROPERTY TypeToken : t_medium_string
GET
                    TypeToken := 'UIRadio';
                  
END_GET
END_PROPERTY

PROPERTY UIOrientation : t_ui_orientation
GET
                    UIOrientation := lUIOrientation;
                  
END_GET
SET
                    IF ((lEnableUIOrientation) AND
	(UIOrientation<>cUIOrientationNone)) THEN
	lUIOrientation := UIOrientation;
END_IF

                  
END_SET
END_PROPERTY

PROPERTY UMFS : BOOL
GET
                    UMFS := ((SafetyCANOpen) AND
	(lInputSafetyHardwiredA.Value) AND
	(lInputSafetyHardwiredB.Value));
	
                  
END_GET
END_PROPERTY

PROPERTY TwistlockUnlock : BOOL
GET
                    TwistlockUnlock := FALSE;

IF (Active) THEN
	TwistlockUnlock := lControllerUInterfaceRadio.TwistlockUnlock;
END_IF

                  
END_GET
END_PROPERTY

PROPERTY ZeroSteerTargetAngle : BOOL
GET
                    ZeroSteerTargetAngle := FALSE;

IF (Active) THEN
	ZeroSteerTargetAngle := lControllerUInterfaceRadio.ZeroSteerTargetAngle;
END_IF

                  
END_GET
END_PROPERTY

PROPERTY EnableBatteryPack : BOOL
GET
                    EnableBatteryPack := lControllerUInterfaceRadio.EnableBatteryPack;

                  
END_GET
END_PROPERTY
END_FUNCTION_BLOCK

FUNCTION_BLOCK UInterfaceDual EXTENDS UInterface
  VAR
    lUInterfaceA : REFERENCE TO UInterface;
    lUInterfaceB : REFERENCE TO UInterface;
    lSwitching : BOOL := FALSE;
    lSwitchTimer : t_timer;
  END_VAR

            ;
          

METHOD initialize
                  SUPER^.initialize();

lUInterfaceA.Resolved REF= THIS^;
lUInterfaceB.Resolved REF= THIS^;
	
lUInterfaceId := cUIIDNone;

lSwitching := FALSE;

lSwitchTimer.lPeriod := T#10s;
lSwitchTimer.initialize();
lSwitchTimer.lEnable := FALSE;

lUInterfaceA.lSingleMode :=FALSE;
lUInterfaceB.lSingleMode :=FALSE;

                
END_METHOD

METHOD operator
                  lDiagnostic := _Diagnostic;
_Diagnostic := cUInterfaceDiagnosticOK;

lUInterfaceA.operator();
lUInterfaceB.operator();

IF ((lUInterfaceA.UIMode<=cUIModeSlave) AND (lUInterfaceA.lReady)) THEN
	CASE (lUInterfaceB.UIMode) OF
		cUIModeInoperable:
			lUInterfaceA.UIMode := cUIModeSingle;
		cUIModeSlave:
			lUInterfaceA.UIMode := cUIModeSlave;
			lUInterfaceB.UIMode := cUIModeMaster;
		cUIModeSingle:
			lUInterfaceA.UIMode := cUIModeSlave;
			lUInterfaceB.UIMode := cUIModeMaster;
		cUIModeMaster:
			lUInterfaceA.UIMode := cUIModeSlave;
			lUInterfaceB.UIMode := cUIModeMaster;
	END_CASE
END_IF

IF ((lUInterfaceB.UIMode<=cUIModeSlave) AND (lUInterfaceB.lReady)) THEN
	CASE (lUInterfaceA.UIMode) OF
		cUIModeInoperable:
			lUInterfaceB.UIMode := cUIModeSingle;
		cUIModeSlave:
			lUInterfaceB.UIMode := cUIModeSlave;
			lUInterfaceA.UIMode := cUIModeMaster;
		cUIModeSingle:
			lUInterfaceB.UIMode := cUIModeSlave;
			lUInterfaceA.UIMode := cUIModeMaster;
		cUIModeMaster:
			lUInterfaceB.UIMode := cUIModeSlave;
			lUInterfaceA.UIMode := cUIModeMaster;
	END_CASE
END_IF

IF ((lUInterfaceB.UIMode=cUIModeInoperable) AND (lUInterfaceA.UIMode=cUIModeMaster)) THEN
	lUInterfaceA.UIMode := cUIModeSingle;
END_IF
IF ((lUInterfaceA.UIMode=cUIModeInoperable) AND (lUInterfaceB.UIMode=cUIModeMaster)) THEN
	lUInterfaceB.UIMode := cUIModeSingle;
END_IF

lReady := (((lUInterfaceA.lReady) AND (lUInterfaceB.UIMode=cUIModeInoperable)) OR
	((lUInterfaceB.lReady) AND (lUInterfaceA.UIMode=cUIModeInoperable)) OR
	((lUInterfaceA.lReady) AND (lUInterfaceB.lReady)));

IF (NOT(lReady)) THEN
	Diagnostic := cUInterfaceDiagnosticNotReady;

	lAlarmUInterfaceNotReady.trigger(FALSE);
END_IF

lSwitchTimer.operator();
lSwitching := ((lSwitchTimer.Enable) AND (NOT(lSwitchTimer.Expired)));
lSwitchTimer.Enable := lSwitching;

IF (NOT(lSwitching)) THEN
	lUInterfaceA.UIModeRequest := FALSE;
	lUInterfaceB.UIModeRequest := FALSE;
END_IF

                
END_METHOD

METHOD uiModeHandler
  VAR_INPUT
    id : t_ui_id;
  END_VAR
                  CASE id OF
	cUIIdA:
		IF ((lUInterfaceA.UIMode=cUIModeSlave) AND (NOT(lSwitching))) THEN
			lSwitching := TRUE;
			lSwitchTimer.Enable := TRUE;
			lSwitchTimer.reset();
			
			lUInterfaceB.UIModeRequest := TRUE;
		END_IF

		IF ((lUInterfaceA.UIMode=cUIModeMaster) AND (lSwitching)) THEN
			lSwitching := FALSE;
			lSwitchTimer.Enable := FALSE;
			lUInterfaceA.UIMode := cUIModeSlave;
			lUInterfaceB.UIMode := cUIModeMaster;
		END_IF

	cUIIdB:
		IF ((lUInterfaceB.UIMode=cUIModeSlave) AND (NOT(lSwitching))) THEN
			lSwitching := TRUE;
			lSwitchTimer.Enable := TRUE;
			lSwitchTimer.reset();

			lUInterfaceA.UIModeRequest := TRUE;
		END_IF

		IF ((lUInterfaceB.UIMode=cUIModeMaster) AND (lSwitching)) THEN
			lSwitching := FALSE;
			lSwitchTimer.Enable := FALSE;
			lUInterfaceB.UIMode := cUIModeSlave;
			lUInterfaceA.UIMode := cUIModeMaster;
		END_IF
END_CASE
                
END_METHOD

PROPERTY Active : BOOL
GET
                    Active := (lUInterfaceA.Active) OR (lUInterfaceB.Active);

                  
END_GET
END_PROPERTY

PROPERTY AutomationRequest : t_prog_mov_code
GET
                    AutomationRequest := cProgMovCodeNone;

IF (lUInterfaceA.Active) THEN
	AutomationRequest := lUInterfaceA.AutomationRequest;
END_IF
IF (lUInterfaceB.Active) THEN
	AutomationRequest := lUInterfaceB.AutomationRequest;
END_IF
                  
END_GET
END_PROPERTY

PROPERTY AutomationStart : BOOL
GET
                    AutomationStart := FALSE;

IF (lUInterfaceA.Active) THEN
	AutomationStart := lUInterfaceA.AutomationStart;
END_IF
IF (lUInterfaceB.Active) THEN
	AutomationStart := lUInterfaceB.AutomationStart;
END_IF

                  
END_GET
END_PROPERTY

(* {attribute 'monitoring' := 'call'} *)
PROPERTY ConfigurationJoystickInputPresent : BOOL
GET
                    ConfigurationJoystickInputPresent := FALSE;

IF (lUInterfaceA.Active) THEN
	ConfigurationJoystickInputPresent := lUInterfaceA.ConfigurationJoystickInputPresent;
END_IF
IF (lUInterfaceB.Active) THEN
	ConfigurationJoystickInputPresent := lUInterfaceB.ConfigurationJoystickInputPresent;
END_IF

                  
END_GET
END_PROPERTY

PROPERTY Emgy : BOOL
GET
                    Emgy := lUInterfaceA.Emgy AND lUInterfaceB.Emgy;

IF (lUInterfaceA.UIMode=cUIModeInoperable) THEN
	Emgy := lUInterfaceB.Emgy;
END_IF
IF (lUInterfaceB.UIMode=cUIModeInoperable) THEN
	Emgy := lUInterfaceA.Emgy;
END_IF
                  
END_GET
END_PROPERTY

PROPERTY Estop : BOOL
GET
                    Estop := lUInterfaceA.Estop AND lUInterfaceB.Estop;

IF (lUInterfaceA.UIMode=cUIModeInoperable) THEN
	Estop := lUInterfaceB.Estop;
END_IF
IF (lUInterfaceB.UIMode=cUIModeInoperable) THEN
	Estop := lUInterfaceA.Estop;
END_IF

                  
END_GET
END_PROPERTY

PROPERTY FunctionalModeRequest : t_functional_mode
GET
                    FunctionalModeRequest := cFunctionalModeAny;

IF (lUInterfaceA.Active) THEN
	FunctionalModeRequest := lUInterfaceA.FunctionalModeRequest;
END_IF
IF (lUInterfaceB.Active) THEN
	FunctionalModeRequest := lUInterfaceB.FunctionalModeRequest;
END_IF
                  
END_GET
END_PROPERTY

PROPERTY Horn : BOOL
GET
                    Horn := (lUInterfaceA.Horn) OR (lUInterfaceB.Horn);
                  
END_GET
END_PROPERTY

PROPERTY IsBeginner : BOOL
GET
                    IsBeginner := FALSE;

IF (lUInterfaceA.Active) THEN
	IsBeginner := lUInterfaceA.IsBeginner;
END_IF
IF (lUInterfaceB.Active) THEN
	IsBeginner := lUInterfaceB.IsBeginner;
END_IF
                  
END_GET
END_PROPERTY

PROPERTY IsSlow : BOOL
GET
                    IsSlow := FALSE;

IF (lUInterfaceA.Active) THEN
	IsSlow := lUInterfaceA.IsSlow;
END_IF
IF (lUInterfaceB.Active) THEN
	IsSlow := lUInterfaceB.IsSlow;
END_IF
                  
END_GET
END_PROPERTY

(* {attribute 'monitoring' := 'call'} *)
PROPERTY JoystickInputPresent : BOOL
GET
                    JoystickInputPresent := FALSE;

IF (lUInterfaceA.Active) THEN
	JoystickInputPresent := lUInterfaceA.JoystickInputPresent;
END_IF
IF (lUInterfaceB.Active) THEN
	JoystickInputPresent := lUInterfaceB.JoystickInputPresent;
END_IF
                  
END_GET
END_PROPERTY

PROPERTY Lift : t_percentage
GET
                    Lift := 0;

IF (lUInterfaceA.Active) THEN
	Lift := lUInterfaceA.Lift;
END_IF
IF (lUInterfaceB.Active) THEN
	Lift := lUInterfaceB.Lift;
END_IF
                  
END_GET
END_PROPERTY

PROPERTY LiftBalanceAB : t_percentage
GET
                    LiftBalanceAB := 0;

IF (lUInterfaceA.Active) THEN
	LiftBalanceAB := lUInterfaceA.LiftBalanceAB;
END_IF
IF (lUInterfaceB.Active) THEN
	LiftBalanceAB := lUInterfaceB.LiftBalanceAB;
END_IF
                  
END_GET
END_PROPERTY

PROPERTY LiftBalanceAD : t_percentage
GET
                    LiftBalanceAD := 0;

IF (lUInterfaceA.Active) THEN
	LiftBalanceAD := lUInterfaceA.LiftBalanceAD;
END_IF
IF (lUInterfaceB.Active) THEN
	LiftBalanceAD := lUInterfaceB.LiftBalanceAD;
END_IF
                  
END_GET
END_PROPERTY

(* {attribute 'monitoring' := 'call'} *)
PROPERTY LiftJoystickInputPresent : BOOL
GET
                    LiftJoystickInputPresent := FALSE;

IF (lUInterfaceA.Active) THEN
	LiftJoystickInputPresent := lUInterfaceA.LiftJoystickInputPresent;
END_IF
IF (lUInterfaceB.Active) THEN
	LiftJoystickInputPresent := lUInterfaceB.LiftJoystickInputPresent;
END_IF

                  
END_GET
END_PROPERTY

PROPERTY OperatingMethodRequest : t_operating_method
GET
                    OperatingMethodRequest := cOperatingMethodNone;

IF (lUInterfaceA.Active) THEN
	OperatingMethodRequest := lUInterfaceA.OperatingMethodRequest;
END_IF
IF (lUInterfaceB.Active) THEN
	OperatingMethodRequest := lUInterfaceB.OperatingMethodRequest;
END_IF
                  
END_GET
END_PROPERTY

PROPERTY Override : BOOL
GET
                    Override := FALSE;
 
IF (lUInterfaceA.Active) THEN
	Override := lUInterfaceA.Override;
END_IF
IF (lUInterfaceB.Active) THEN
	Override := lUInterfaceB.Override;
END_IF
                  
END_GET
END_PROPERTY

PROPERTY SideshiftAB : t_percentage
GET
                    SideshiftAB := 0;

IF (lUInterfaceA.Active) THEN
	SideshiftAB := lUInterfaceA.SideshiftAB;
END_IF
IF (lUInterfaceB.Active) THEN
	SideshiftAB := lUInterfaceB.SideshiftAB;
END_IF
                  
END_GET
END_PROPERTY

PROPERTY SideshiftCD : t_percentage
GET
                    SideshiftCD := 0;

IF (lUInterfaceA.Active) THEN
	SideshiftCD := lUInterfaceA.SideshiftCD;
END_IF
IF (lUInterfaceB.Active) THEN
	SideshiftCD := lUInterfaceB.SideshiftCD;
END_IF
                  
END_GET
END_PROPERTY

PROPERTY SlowFactor : REAL
GET
                    SlowFactor := 1.0;

IF (lUInterfaceA.Active) THEN
	SlowFactor := lUInterfaceA.SlowFactor;
END_IF
IF (lUInterfaceB.Active) THEN
	SlowFactor := lUInterfaceB.SlowFactor;
END_IF
                  
END_GET
END_PROPERTY

PROPERTY SpreaderTelescopingExtend : BOOL
GET
                    SpreaderTelescopingExtend := FALSE;

IF (lUInterfaceA.Active) THEN
	SpreaderTelescopingExtend := lUInterfaceA.SpreaderTelescopingExtend;
END_IF
IF (lUInterfaceB.Active) THEN
	SpreaderTelescopingExtend := lUInterfaceB.SpreaderTelescopingExtend;
END_IF
                  
END_GET
END_PROPERTY

PROPERTY SpreaderTelescopingRetract : BOOL
GET
                    SpreaderTelescopingRetract := FALSE;

IF (lUInterfaceA.Active) THEN
	SpreaderTelescopingRetract := lUInterfaceA.SpreaderTelescopingRetract;
END_IF
IF (lUInterfaceB.Active) THEN
	SpreaderTelescopingRetract := lUInterfaceB.SpreaderTelescopingRetract;
END_IF
                  
END_GET
END_PROPERTY

PROPERTY Steer : t_percentage
GET
                    Steer := 0;

IF (lUInterfaceA.Active) THEN
	Steer := lUInterfaceA.Steer;
END_IF
IF (lUInterfaceB.Active) THEN
	Steer := lUInterfaceB.Steer;
END_IF
                  
END_GET
END_PROPERTY

PROPERTY SteerModeRequest : t_steer_mode
GET
                    SteerModeRequest := cSteerModeNone;

IF (lUInterfaceA.Active) THEN
	SteerModeRequest := lUInterfaceA.SteerModeRequest;
END_IF
IF (lUInterfaceB.Active) THEN
	SteerModeRequest := lUInterfaceB.SteerModeRequest;
END_IF
                  
END_GET
END_PROPERTY

PROPERTY Stop : BOOL
GET
                    Stop := lUInterfaceA.Stop AND lUInterfaceB.Stop;

IF (lUInterfaceA.UIMode=cUIModeInoperable) THEN
	Stop := lUInterfaceB.Stop;
END_IF
IF (lUInterfaceB.UIMode=cUIModeInoperable) THEN
	Stop := lUInterfaceA.Stop;
END_IF
                  
END_GET
END_PROPERTY

(* {attribute 'monitoring' := 'call'} *)
PROPERTY Switching : BOOL
GET
                    Switching := lSwitching;
                  
END_GET
END_PROPERTY

PROPERTY Topbeam : t_percentage
GET
                    Topbeam := 0;

IF (lUInterfaceA.Active) THEN
	Topbeam := lUInterfaceA.Topbeam;
END_IF
IF (lUInterfaceB.Active) THEN
	Topbeam := lUInterfaceB.Topbeam;
END_IF
                  
END_GET
END_PROPERTY

(* {attribute 'monitoring' := 'call'} *)
PROPERTY Travel : t_percentage
GET
                    Travel := 0;

IF (lUInterfaceA.Active) THEN
	Travel := lUInterfaceA.Travel;
END_IF
IF (lUInterfaceB.Active) THEN
	Travel := lUInterfaceB.Travel;
END_IF
                  
END_GET
END_PROPERTY

(* {attribute 'monitoring' := 'call'} *)
PROPERTY TravelJoystickInputPresent : BOOL
GET
                    TravelJoystickInputPresent := FALSE;

IF (lUInterfaceA.Active) THEN
	TravelJoystickInputPresent := lUInterfaceA.TravelJoystickInputPresent;
END_IF
IF (lUInterfaceB.Active) THEN
	TravelJoystickInputPresent := lUInterfaceB.TravelJoystickInputPresent;
END_IF

                  
END_GET
END_PROPERTY

PROPERTY TriggerRespond : t_ui_id
SET
                    uiModeHandler(TriggerRespond);

                  
END_SET
END_PROPERTY

PROPERTY TwistlockLock : BOOL
GET
                    TwistlockLock := FALSE;
 
IF (lUInterfaceA.Active) THEN
	TwistlockLock := lUInterfaceA.TwistlockLock;
END_IF
IF (lUInterfaceB.Active) THEN
	TwistlockLock := lUInterfaceB.TwistlockLock;
END_IF
                  
END_GET
END_PROPERTY

PROPERTY TwistlockUnlock : BOOL
GET
                    TwistlockUnlock := FALSE;
 
IF (lUInterfaceA.Active) THEN
	TwistlockUnlock := lUInterfaceA.TwistlockUnlock;
END_IF
IF (lUInterfaceB.Active) THEN
	TwistlockUnlock := lUInterfaceB.TwistlockUnlock;
END_IF
                  
END_GET
END_PROPERTY

PROPERTY TypeToken : t_medium_string
GET
                    TypeToken := 'UIDual';
                  
END_GET
END_PROPERTY

PROPERTY UIEventCodeRequest : t_ui_event_code
GET
                    UIEventCodeRequest := cUIEventCodeNone;
 
IF (lUInterfaceA.Active) THEN
	UIEventCodeRequest := lUInterfaceA.UIEventCodeRequest;
END_IF
IF (lUInterfaceB.Active) THEN
	UIEventCodeRequest := lUInterfaceB.UIEventCodeRequest;
END_IF
                  
END_GET
END_PROPERTY

PROPERTY UIMode : t_ui_mode
GET
                    UIMode := cUIModeInoperable;

                  
END_GET
SET
                    
                  
END_SET
END_PROPERTY

PROPERTY UInterfaceA : REFERENCE TO UInterface
GET
                    UInterfaceA ref= lUInterfaceA;
                  
END_GET
SET
                    lUInterfaceA REF= UInterfaceA;

                  
END_SET
END_PROPERTY

PROPERTY UInterfaceB : REFERENCE TO UInterface
GET
                    UInterfaceB ref= lUInterfaceB;
                  
END_GET
SET
                    lUInterfaceB REF= UInterfaceB;

                  
END_SET
END_PROPERTY

PROPERTY UInterfaceId : t_ui_id
GET
                    UInterfaceId := lUInterfaceId;

IF (lUInterfaceA.Active) THEN
	UInterfaceId := lUInterfaceA.UInterfaceId;
END_IF
IF (lUInterfaceB.Active) THEN
	UInterfaceId := lUInterfaceB.UInterfaceId;
END_IF
                  
END_GET
END_PROPERTY

PROPERTY UMFS : BOOL
GET
                    IF (lUInterfaceA.Active) THEN
	UMFS := lUInterfaceA.UMFS;
END_IF
IF (lUInterfaceB.Active) THEN
	UMFS := lUInterfaceB.UMFS;
END_IF

(*
UMFS := lUInterfaceA.UMFS AND lUInterfaceB.UMFS;

IF (lUInterfaceA.UIMode=cUIModeInoperable) THEN
	UMFS := lUInterfaceB.UMFS;
END_IF
IF (lUInterfaceB.UIMode=cUIModeInoperable) THEN
	UMFS := lUInterfaceA.UMFS;
END_IF
*)
                  
END_GET
END_PROPERTY

PROPERTY ZeroSteerTargetAngle : BOOL
GET
                    ZeroSteerTargetAngle := FALSE;
 
IF (lUInterfaceA.Active) THEN
	ZeroSteerTargetAngle := lUInterfaceA.ZeroSteerTargetAngle;
END_IF
IF (lUInterfaceB.Active) THEN
	ZeroSteerTargetAngle := lUInterfaceB.ZeroSteerTargetAngle;
END_IF
                  
END_GET
END_PROPERTY

(* {attribute 'monitoring' := 'call'} *)
PROPERTY EnableBatteryPack : BOOL
GET
                    EnableBatteryPack := ((lUInterfaceA.EnableBatteryPack) AND (lUInterfaceB.EnableBatteryPack));

IF (lUInterfaceA.UIMode=cUIModeInoperable) THEN
	EnableBatteryPack := lUInterfaceB.EnableBatteryPack;
END_IF
IF (lUInterfaceB.UIMode=cUIModeInoperable) THEN
	EnableBatteryPack := lUInterfaceA.EnableBatteryPack;
END_IF

                  
END_GET
END_PROPERTY
END_FUNCTION_BLOCK

FUNCTION_BLOCK UInterfacePLC EXTENDS UInterface
  VAR
    lPackChannelUInterface : PackChannelUInterfacePLC;
    lUIRRouter : UIRRouter;
    lUIEventCodeRequest : ValueObjectEnumType;
    lSteerModeRequest : ValueObjectEnumType;
    lOperatingMethodRequest : ValueObjectEnumType;
    lFunctionalModeRequest : ValueObjectEnumType;
    lAutomationRequest : ValueObjectEnumType;
    lUIModeResponse : ValueObjectBoolChange;
    lIsBeginner : ValueObjectBool;
    lOverride : ValueObjectBool;
  END_VAR

            ;
          

METHOD initialize
                  lUIEventCodeRequest.EnumType := cEnumTypeUiEventCode;
lUIEventCodeRequest.initializeValueObjectOp(OpSelf,'EventCodeReq','Event code request','',cValueStyleConfigurable);

lSteerModeRequest.EnumType := cEnumTypeSteerMode;
lSteerModeRequest.initializeValueObjectOp(OpSelf,'SteerModeReq','Steer mode request','',cValueStyleConfigurable);

lOperatingMethodRequest.EnumType := cEnumTypeOperatingMethod;
lOperatingMethodRequest.initializeValueObjectOp(OpSelf,'OpMethReq','Operating method request','',cValueStyleConfigurable);

lFunctionalModeRequest.EnumType := cEnumTypeFunctionalMode;
lFunctionalModeRequest.initializeValueObjectOp(OpSelf,'FuncModeReq','Functional mode request','',cValueStyleConfigurable);

lAutomationRequest.EnumType := cEnumTypeProgMovCode;
lAutomationRequest.initializeValueObjectOp(OpSelf,'AutomationReq','Automation request','',cValueStyleConfigurable);

lIsBeginner.initializeValueObjectOp(OpSelf,'IsBeginner','Forces user to beginner mode','',cValueStyleConfigurable);
lUIModeResponse.initializeValueObjectOp(OpSelf,'UIModeResp','UI mode response','',cValueStyleConfigurable);
lOverride.initializeValueObjectOp(OpSelf,'Override','Override mode is active','',cValueStyleConfigurable);

registerOperational(ADR(lPackChannelUInterface));
registerNonOperational(ADR(lUIRRouter));

SUPER^.initialize();

                
END_METHOD

METHOD initializeUInterfacePLC
  VAR_INPUT
    packSystem : REFERENCE TO PackSystemPLC;
    packMovement : REFERENCE TO PackMovementPLC;
    packReportable : REFERENCE TO PackReportablePLC;
    packSpreader : REFERENCE TO PackSpreader;
    packUICommand : REFERENCE TO PackUICommandPLC;
    packProvider : REFERENCE TO PackProvider;
  END_VAR
                  lPackChannelUInterface.initializePackChannelUInterface(packSystem,
	packMovement,
	packReportable,
	packSpreader,
	packUICommand,
	packProvider);

                
END_METHOD

PROPERTY FunctionalModeRequest : t_functional_mode
GET
                    FunctionalModeRequest := cFunctionalModeAny;

IF (Active) THEN
	FunctionalModeRequest := lFunctionalModeRequest.Value;
END_IF

                  
END_GET
SET
                    lFunctionalModeRequest.Value := FunctionalModeRequest;

                  
END_SET
END_PROPERTY

PROPERTY IsBeginner : BOOL
GET
                    IsBeginner := lIsBeginner.Value;

                  
END_GET
SET
                    lIsBeginner.Value := IsBeginner;

                  
END_SET
END_PROPERTY

PROPERTY UIOrientation : t_ui_orientation
SET
                    
                  
END_SET
END_PROPERTY

PROPERTY OperatingMethodRequest : t_operating_method
GET
                    OperatingMethodRequest := cOperatingMethodNone;

IF (Active) THEN
	OperatingMethodRequest := lOperatingMethodRequest.Value;
END_IF
                  
END_GET
SET
                    lOperatingMethodRequest.Value := OperatingMethodRequest;

                  
END_SET
END_PROPERTY

PROPERTY Override : BOOL
GET
                    Override := FALSE;

IF (Active) THEN
	Override := lOverride.Value;
END_IF

                  
END_GET
SET
                    lOverride.Value := Override;

                  
END_SET
END_PROPERTY

PROPERTY SteerModeRequest : t_steer_mode
GET
                    SteerModeRequest := cSteerModeNone;

IF (Active) THEN
	SteerModeRequest := lSteerModeRequest.Value;
END_IF
                  
END_GET
SET
                    lSteerModeRequest.Value := SteerModeRequest;

                  
END_SET
END_PROPERTY

PROPERTY InputMode : t_input_mode
SET
                    

                  
END_SET
END_PROPERTY

PROPERTY UIRRouter : REFERENCE TO UIRRouter
GET
                    UIRRouter ref= lUIRRouter;
                  
END_GET
END_PROPERTY

PROPERTY AutomationRequest : t_prog_mov_code
GET
                    AutomationRequest := cProgMovCodeNone;

IF (Active) THEN
	AutomationRequest := lAutomationRequest.Value;
END_IF
                  
END_GET
SET
                    lAutomationRequest.Value := AutomationRequest;

                  
END_SET
END_PROPERTY

PROPERTY UIEventCodeRequest : t_ui_event_code
GET
                    UIEventCodeRequest := cUIEventCodeNone;

IF (Active) THEN
	UIEventCodeRequest := lUIEventCodeRequest.Value;
END_IF
                  
END_GET
SET
                    lUIEventCodeRequest.Value := UIEventCodeRequest;

                  
END_SET
END_PROPERTY

(* {attribute 'monitoring' := 'call'} *)
PROPERTY UIModeResponse : BOOL
GET
                    UIModeResponse := lUIModeResponse.Rising;


                  
END_GET
SET
                    lUIModeResponse.Value := UIModeResponse;

                  
END_SET
END_PROPERTY
END_FUNCTION_BLOCK

FUNCTION_BLOCK CANOpenMasterDrivePrimary EXTENDS CANOpenMaster
  VAR
    lSteerAngleA : ControllerRotaryEncoderRange;
    lSteerAngleB : ControllerRotaryEncoderRange;
    lSteerAngleC : ControllerRotaryEncoderRange;
    lSteerAngleD : ControllerRotaryEncoderRange;
    lSteerA : ControllerMotor;
    lSteerB : ControllerMotor;
    lSteerC : ControllerMotor;
    lSteerD : ControllerMotor;
  END_VAR

            ;
          

METHOD initialize
                  Name := 'CANBusDrive';

lSteerA.lTypeSteer := TRUE;
lSteerB.lTypeSteer := TRUE;
lSteerC.lTypeSteer := TRUE;
lSteerD.lTypeSteer := TRUE;

lSteerAngleA.lTypeSteer := TRUE;
lSteerAngleB.lTypeSteer := TRUE;
lSteerAngleC.lTypeSteer := TRUE;
lSteerAngleD.lTypeSteer := TRUE;

lSteerAngleA.Name := 'cSteerAngleA';
lSteerAngleA.SubSystem := cSubsystemSteerA;
lSteerAngleA.NetworkId := 2;
registerOperational(ADR(lSteerAngleA));

lSteerAngleB.Name := 'cSteerAngleB';
lSteerAngleB.SubSystem := cSubsystemSteerB;
lSteerAngleB.NetworkId := 2;
registerOperational(ADR(lSteerAngleB));

lSteerAngleC.Name := 'cSteerAngleC';
lSteerAngleC.SubSystem := cSubsystemSteerC;
lSteerAngleC.NetworkId := 2;
registerOperational(ADR(lSteerAngleC));

lSteerAngleD.Name := 'cSteerAngleD';
lSteerAngleD.SubSystem := cSubsystemSteerD;
lSteerAngleD.NetworkId := 2;
registerOperational(ADR(lSteerAngleD));

lSteerA.Name := 'cSteerA';
lSteerA.SubSystem := cSubsystemSteerA;
lSteerA.NetworkId := 2;
registerOperational(ADR(lSteerA));

lSteerB.Name := 'cSteerB';
lSteerB.SubSystem := cSubsystemSteerB;
lSteerB.NetworkId := 2;
registerOperational(ADR(lSteerB));

lSteerC.Name := 'cSteerC';
lSteerC.SubSystem := cSubsystemSteerC;
lSteerC.NetworkId := 2;
registerOperational(ADR(lSteerC));

lSteerD.Name := 'cSteerD';
lSteerD.SubSystem := cSubsystemSteerD;
lSteerD.NetworkId := 2;
registerOperational(ADR(lSteerD));

SUPER^.initialize();
SubSystem := cSubsystemCANBusDrive;

lOperationalSystemStateScope := cSystemStateGoOperational;
lAllowableUpSystemStateScope := cSystemStatePoweringUp;
lSystemControlRecovery := cSystemControlStop;

lBusPower.OutputSystemState := cSystemStatePoweringDown;
lEstopOnNodeState := FALSE;

                
END_METHOD

(* {attribute 'monitoring' := 'call'} *)
PROPERTY SteerAngleB : REFERENCE TO ControllerRotaryEncoderRange
GET
                    SteerAngleB REF= lSteerAngleB;

                  
END_GET
END_PROPERTY

(* {attribute 'monitoring' := 'call'} *)
PROPERTY SteerAngleD : REFERENCE TO ControllerRotaryEncoderRange
GET
                    SteerAngleD REF= lSteerAngleD;

                  
END_GET
END_PROPERTY

(* {attribute 'monitoring' := 'call'} *)
PROPERTY SteerA : REFERENCE TO ControllerMotor
GET
                    SteerA REF= lSteerA;

                  
END_GET
END_PROPERTY

(* {attribute 'monitoring' := 'call'} *)
PROPERTY SteerB : REFERENCE TO ControllerMotor
GET
                    SteerB REF= lSteerB;

                  
END_GET
END_PROPERTY

(* {attribute 'monitoring' := 'call'} *)
PROPERTY SteerC : REFERENCE TO ControllerMotor
GET
                    SteerC REF= lSteerC;

                  
END_GET
END_PROPERTY

(* {attribute 'monitoring' := 'call'} *)
PROPERTY SteerAngleA : REFERENCE TO ControllerRotaryEncoderRange
GET
                    SteerAngleA REF= lSteerAngleA;

                  
END_GET
END_PROPERTY

(* {attribute 'monitoring' := 'call'} *)
PROPERTY SteerAngleC : REFERENCE TO ControllerRotaryEncoderRange
GET
                    SteerAngleC REF= lSteerAngleC;

                  
END_GET
END_PROPERTY

(* {attribute 'monitoring' := 'call'} *)
PROPERTY SteerD : REFERENCE TO ControllerMotor
GET
                    SteerD REF= lSteerD;

                  
END_GET
END_PROPERTY
END_FUNCTION_BLOCK

FUNCTION_BLOCK CANOpenMasterSystemPrimary EXTENDS CANOpenMaster
  VAR
    lSecondaryPowerSupplyA : ControllerSecondaryPowerSupply;
    lSecondaryPowerSupplyB : ControllerSecondaryPowerSupply;
  END_VAR

            ;
          

METHOD initialize
                  Name := 'CANBusSystem';

lSecondaryPowerSupplyA.Name := 'cSecondaryA';
lSecondaryPowerSupplyA.SubSystem := cSubsystemSecondary;
lSecondaryPowerSupplyA.NetworkId := 1;
lSecondaryPowerSupplyA.initializeSecondary(gSystemPrimary.SecondaryPowerSupply);
registerOperational(ADR(lSecondaryPowerSupplyA));

